LIN {X 0,Y 357.661,Z 442.016,A -85,B 0,C 180,E1 -17550,E2 -17550} C_VEL
LIN {X 0,Y 357.419,Z 441.985,A -85,B 0,C 180,E1 -17551.127,E2 -17551.127} C_VEL
LIN {X 0,Y 356.749,Z 441.848,A -85,B 0,C 180,E1 -17552.258,E2 -17552.258} C_VEL
LIN {X 0,Y 355.709,Z 441.54,A -85,B 0,C 180,E1 -17553.398,E2 -17553.398} C_VEL
LIN {X 0,Y 354.333,Z 441.001,A -85,B 0,C 180,E1 -17554.55,E2 -17554.55} C_VEL
LIN {X 0,Y 352.777,Z 440.106,A -85,B 0,C 180,E1 -17555.717,E2 -17555.717} C_VEL
LIN {X 0,Y 351.014,Z 438.819,A -85,B 0,C 180,E1 -17556.9,E2 -17556.9} C_VEL
LIN {X 0,Y 348.295,Z 436.243,A -85,B 0,C 180,E1 -17558.613,E2 -17558.613} C_VEL
LIN {X 0,Y 346.111,Z 434.166,A -85,B 0,C 180,E1 -17559.779,E2 -17559.779} C_VEL
LIN {X 0,Y 342.714,Z 431.618,A -85,B 0,C 180,E1 -17561.14,E2 -17561.14} C_VEL
LIN {X 0,Y 338.593,Z 427.938,A -85,B 0,C 180,E1 -17562.698,E2 -17562.698} C_VEL
LIN {X 0,Y 333.67,Z 423.547,A -85,B 0,C 180,E1 -17564.333,E2 -17564.333} C_VEL
LIN {X 0,Y 327.334,Z 417.343,A -85,B 0,C 180,E1 -17566.207,E2 -17566.207} C_VEL
LIN {X 0,Y 321.069,Z 411.064,A -85,B 0,C 180,E1 -17567.845,E2 -17567.845} C_VEL
LIN {X 0,Y 314.685,Z 404.327,A -85,B 0,C 180,E1 -17569.339,E2 -17569.339} C_VEL
LIN {X 0,Y 306.772,Z 395.528,A -85,B 0,C 180,E1 -17571.006,E2 -17571.006} C_VEL
LIN {X 0,Y 297.489,Z 384.138,A -85,B 0,C 180,E1 -17572.878,E2 -17572.878} C_VEL
LIN {X 0,Y 291.289,Z 375.491,A -85,B 0,C 180,E1 -17574.11,E2 -17574.11} C_VEL
LIN {X 0,Y 286.082,Z 366.576,A -85,B 0,C 180,E1 -17575.163,E2 -17575.163} C_VEL
LIN {X 0,Y 281.303,Z 356.248,A -85,B 0,C 180,E1 -17576.119,E2 -17576.119} C_VEL
LIN {X 0,Y 277.576,Z 348.553,A -85,B 0,C 180,E1 -17576.746,E2 -17576.746} C_VEL
LIN {X 0,Y 277.359,Z 347.437,A -85,B 0,C 180,E1 -17576.824,E2 -17576.824} C_VEL
LIN {X 0,Y 277.268,Z 347.449,A -85,B 0,C 180,E1 -17580.482,E2 -17580.482} C_VEL
LIN {X 0,Y 277.251,Z 347.451,A -85,B 0,C 180,E1 -17583.895,E2 -17583.895} C_VEL
LIN {X 0,Y 277.286,Z 347.444,A -85,B 0,C 180,E1 -17587.466,E2 -17587.466} C_VEL
LIN {X 0,Y 277.238,Z 347.449,A -85,B 0,C 180,E1 -17591.231,E2 -17591.231} C_VEL
LIN {X 0,Y 277.248,Z 347.448,A -85,B 0,C 180,E1 -17595.216,E2 -17595.216} C_VEL
LIN {X 0,Y 277.292,Z 347.445,A -85,B 0,C 180,E1 -17599.495,E2 -17599.495} C_VEL
LIN {X 0,Y 277.288,Z 347.443,A -85,B 0,C 180,E1 -17602.535,E2 -17602.535} C_VEL
LIN {X 0,Y 277.252,Z 347.448,A -85,B 0,C 180,E1 -17606.106,E2 -17606.106} C_VEL
LIN {X 0,Y 277.259,Z 347.45,A -85,B 0,C 180,E1 -17609.539,E2 -17609.539} C_VEL
LIN {X 0,Y 277.359,Z 347.435,A -85,B 0,C 180,E1 -17612.865,E2 -17612.865} C_VEL
LIN {X 0,Y 277.295,Z 347.441,A -85,B 0,C 180,E1 -17616.077,E2 -17616.077} C_VEL
LIN {X 0,Y 277.343,Z 347.433,A -85,B 0,C 180,E1 -17620.767,E2 -17620.767} C_VEL
LIN {X 0,Y 277.433,Z 347.425,A -85,B 0,C 180,E1 -17625.327,E2 -17625.327} C_VEL
LIN {X 0,Y 277.506,Z 347.413,A -85,B 0,C 180,E1 -17629.79,E2 -17629.79} C_VEL
LIN {X 0,Y 277.648,Z 347.4,A -85,B 0,C 180,E1 -17632.73,E2 -17632.73} C_VEL
LIN {X 0,Y 277.82,Z 347.363,A -85,B 0,C 180,E1 -17638.551,E2 -17638.551} C_VEL
LIN {X 0,Y 277.821,Z 347.375,A -85,B 0,C 180,E1 -17641.45,E2 -17641.45} C_VEL
LIN {X 0,Y 277.649,Z 347.399,A -85,B 0,C 180,E1 -17647.272,E2 -17647.272} C_VEL
LIN {X 0,Y 277.507,Z 347.418,A -85,B 0,C 180,E1 -17650.212,E2 -17650.212} C_VEL
LIN {X 0,Y 277.41,Z 347.432,A -85,B 0,C 180,E1 -17654.676,E2 -17654.676} C_VEL
LIN {X 0,Y 277.324,Z 347.439,A -85,B 0,C 180,E1 -17659.236,E2 -17659.236} C_VEL
LIN {X 0,Y 277.298,Z 347.446,A -85,B 0,C 180,E1 -17663.924,E2 -17663.924} C_VEL
LIN {X 0,Y 277.306,Z 347.44,A -85,B 0,C 180,E1 -17666.283,E2 -17666.283} C_VEL
LIN {X 0,Y 276.643,Z 347.527,A -85,B 0,C 180,E1 -17667.495,E2 -17667.495} C_VEL
LIN {X 0,Y 273.723,Z 347.889,A -85,B 0,C 180,E1 -17669.467,E2 -17669.467} C_VEL
LIN {X 0,Y 271.283,Z 348.334,A -85,B 0,C 180,E1 -17671.069,E2 -17671.069} C_VEL
LIN {X 0,Y 270.308,Z 348.795,A -85,B 0,C 180,E1 -17672.309,E2 -17672.309} C_VEL
LIN {X 0,Y 270.268,Z 348.983,A -85,B 0,C 180,E1 -17672.729,E2 -17672.729} C_VEL
LIN {X 0,Y 270.568,Z 351.115,A -85,B 0,C 180,E1 -17676.687,E2 -17676.687} C_VEL
LIN {X 0,Y 270.931,Z 353.364,A -85,B 0,C 180,E1 -17680.43,E2 -17680.43} C_VEL
LIN {X 0,Y 271.228,Z 355.986,A -85,B 0,C 180,E1 -17684.397,E2 -17684.397} C_VEL
LIN {X 0,Y 271.177,Z 358.336,A -85,B 0,C 180,E1 -17687.637,E2 -17687.637} C_VEL
LIN {X 0,Y 270.855,Z 361.072,A -85,B 0,C 180,E1 -17691.118,E2 -17691.118} C_VEL
LIN {X 0,Y 270.211,Z 364.37,A -85,B 0,C 180,E1 -17695.096,E2 -17695.096} C_VEL
LIN {X 0,Y 269.608,Z 368.108,A -85,B 0,C 180,E1 -17699.343,E2 -17699.343} C_VEL
LIN {X 0,Y 269.108,Z 371.071,A -85,B 0,C 180,E1 -17702.655,E2 -17702.655} C_VEL
LIN {X 0,Y 269.855,Z 374.098,A -85,B 0,C 180,E1 -17702.867,E2 -17702.867} C_VEL
LIN {X 0,Y 273.605,Z 387.988,A -85,B 0,C 180,E1 -17704.108,E2 -17704.108} C_VEL
LIN {X 0,Y 275.578,Z 397.942,A -85,B 0,C 180,E1 -17705.138,E2 -17705.138} C_VEL
LIN {X 0,Y 276.733,Z 406.314,A -85,B 0,C 180,E1 -17706.103,E2 -17706.103} C_VEL
LIN {X 0,Y 277.56,Z 416.03,A -85,B 0,C 180,E1 -17707.392,E2 -17707.392} C_VEL
LIN {X 0,Y 277.591,Z 422.084,A -85,B 0,C 180,E1 -17708.268,E2 -17708.268} C_VEL
LIN {X 0,Y 275.683,Z 432.23,A -85,B 0,C 180,E1 -17709.87,E2 -17709.87} C_VEL
LIN {X 0,Y 274.223,Z 439.743,A -85,B 0,C 180,E1 -17711.316,E2 -17711.316} C_VEL
LIN {X 0,Y 272.724,Z 447.572,A -85,B 0,C 180,E1 -17713.148,E2 -17713.148} C_VEL
LIN {X 0,Y 271.411,Z 454.11,A -85,B 0,C 180,E1 -17714.993,E2 -17714.993} C_VEL
LIN {X 0,Y 270.443,Z 458.61,A -85,B 0,C 180,E1 -17716.474,E2 -17716.474} C_VEL
LIN {X 0,Y 269.43,Z 464.105,A -85,B 0,C 180,E1 -17718.718,E2 -17718.718} C_VEL
LIN {X 0,Y 268.75,Z 468.433,A -85,B 0,C 180,E1 -17720.973,E2 -17720.973} C_VEL
LIN {X 0,Y 268.431,Z 470.802,A -85,B 0,C 180,E1 -17722.478,E2 -17722.478} C_VEL
LIN {X 0,Y 268.181,Z 473.429,A -85,B 0,C 180,E1 -17724.775,E2 -17724.775} C_VEL
LIN {X 0,Y 268.169,Z 475.056,A -85,B 0,C 180,E1 -17726.995,E2 -17726.995} C_VEL
LIN {X 0,Y 268.184,Z 475.647,A -85,B 0,C 180,E1 -17728.498,E2 -17728.498} C_VEL
LIN {X 0,Y 268.184,Z 475.647,A -85,B 0,C 180,E1 -17731.502,E2 -17731.502} C_VEL
LIN {X 0,Y 268.168,Z 475.056,A -85,B 0,C 180,E1 -17733.005,E2 -17733.005} C_VEL
LIN {X 0,Y 268.227,Z 472.603,A -85,B 0,C 180,E1 -17736.016,E2 -17736.016} C_VEL
LIN {X 0,Y 268.565,Z 469.651,A -85,B 0,C 180,E1 -17738.275,E2 -17738.275} C_VEL
LIN {X 0,Y 269.197,Z 465.66,A -85,B 0,C 180,E1 -17740.53,E2 -17740.53} C_VEL
LIN {X 0,Y 270.047,Z 460.526,A -85,B 0,C 180,E1 -17742.78,E2 -17742.78} C_VEL
LIN {X 0,Y 271.136,Z 455.265,A -85,B 0,C 180,E1 -17744.639,E2 -17744.639} C_VEL
LIN {X 0,Y 272.175,Z 450.324,A -85,B 0,C 180,E1 -17746.116,E2 -17746.116} C_VEL
LIN {X 0,Y 273.369,Z 444.625,A -85,B 0,C 180,E1 -17747.582,E2 -17747.582} C_VEL
LIN {X 0,Y 274.872,Z 436.066,A -85,B 0,C 180,E1 -17749.414,E2 -17749.414} C_VEL
LIN {X 0,Y 276.471,Z 427.889,A -85,B 0,C 180,E1 -17750.848,E2 -17750.848} C_VEL
LIN {X 0,Y 277.757,Z 420.73,A -85,B 0,C 180,E1 -17751.914,E2 -17751.914} C_VEL
LIN {X 0,Y 277.247,Z 411.653,A -85,B 0,C 180,E1 -17753.206,E2 -17753.206} C_VEL
LIN {X 0,Y 276.147,Z 401.415,A -85,B 0,C 180,E1 -17754.465,E2 -17754.465} C_VEL
LIN {X 0,Y 274.464,Z 391.943,A -85,B 0,C 180,E1 -17755.495,E2 -17755.495} C_VEL
LIN {X 0,Y 271.783,Z 380.805,A -85,B 0,C 180,E1 -17756.553,E2 -17756.553} C_VEL
LIN {X 0,Y 269.109,Z 371.049,A -85,B 0,C 180,E1 -17757.383,E2 -17757.383} C_VEL
LIN {X 0,Y 269.703,Z 367.344,A -85,B 0,C 180,E1 -17761.41,E2 -17761.41} C_VEL
LIN {X 0,Y 270.228,Z 364.33,A -85,B 0,C 180,E1 -17764.901,E2 -17764.901} C_VEL
LIN {X 0,Y 270.855,Z 361.042,A -85,B 0,C 180,E1 -17768.882,E2 -17768.882} C_VEL
LIN {X 0,Y 271.18,Z 358.333,A -85,B 0,C 180,E1 -17772.363,E2 -17772.363} C_VEL
LIN {X 0,Y 271.228,Z 355.975,A -85,B 0,C 180,E1 -17775.603,E2 -17775.603} C_VEL
LIN {X 0,Y 270.927,Z 353.357,A -85,B 0,C 180,E1 -17779.569,E2 -17779.569} C_VEL
LIN {X 0,Y 270.546,Z 350.92,A -85,B 0,C 180,E1 -17783.638,E2 -17783.638} C_VEL
LIN {X 0,Y 270.314,Z 349.153,A -85,B 0,C 180,E1 -17786.907,E2 -17786.907} C_VEL
LIN {X 0,Y 270.202,Z 348.332,A -85,B 0,C 180,E1 -17789.13,E2 -17789.13} C_VEL
LIN {X 0,Y 270.265,Z 348.321,A -85,B 0,C 180,E1 -17792.145,E2 -17792.145} C_VEL
LIN {X 0,Y 270.239,Z 348.325,A -85,B 0,C 180,E1 -17795.537,E2 -17795.537} C_VEL
LIN {X 0,Y 270.261,Z 348.32,A -85,B 0,C 180,E1 -17800.241,E2 -17800.241} C_VEL
LIN {X 0,Y 270.377,Z 348.305,A -85,B 0,C 180,E1 -17804.933,E2 -17804.933} C_VEL
LIN {X 0,Y 270.442,Z 348.3,A -85,B 0,C 180,E1 -17809.518,E2 -17809.518} C_VEL
LIN {X 0,Y 270.608,Z 348.275,A -85,B 0,C 180,E1 -17812.538,E2 -17812.538} C_VEL
LIN {X 0,Y 270.787,Z 348.251,A -85,B 0,C 180,E1 -17818.512,E2 -17818.512} C_VEL
LIN {X 0,Y 270.786,Z 348.238,A -85,B 0,C 180,E1 -17821.486,E2 -17821.486} C_VEL
LIN {X 0,Y 270.607,Z 348.276,A -85,B 0,C 180,E1 -17827.46,E2 -17827.46} C_VEL
LIN {X 0,Y 270.441,Z 348.294,A -85,B 0,C 180,E1 -17830.48,E2 -17830.48} C_VEL
LIN {X 0,Y 270.402,Z 348.301,A -85,B 0,C 180,E1 -17835.064,E2 -17835.064} C_VEL
LIN {X 0,Y 270.3,Z 348.309,A -85,B 0,C 180,E1 -17839.755,E2 -17839.755} C_VEL
LIN {X 0,Y 270.236,Z 348.321,A -85,B 0,C 180,E1 -17844.588,E2 -17844.588} C_VEL
LIN {X 0,Y 270.27,Z 348.318,A -85,B 0,C 180,E1 -17847.908,E2 -17847.908} C_VEL
LIN {X 0,Y 270.182,Z 348.328,A -85,B 0,C 180,E1 -17851.347,E2 -17851.347} C_VEL
LIN {X 0,Y 270.213,Z 348.325,A -85,B 0,C 180,E1 -17854.903,E2 -17854.903} C_VEL
LIN {X 0,Y 270.219,Z 348.325,A -85,B 0,C 180,E1 -17858.716,E2 -17858.716} C_VEL
LIN {X 0,Y 270.22,Z 348.325,A -85,B 0,C 180,E1 -17862.548,E2 -17862.548} C_VEL
LIN {X 0,Y 270.201,Z 348.326,A -85,B 0,C 180,E1 -17866.742,E2 -17866.742} C_VEL
LIN {X 0,Y 270.234,Z 348.323,A -85,B 0,C 180,E1 -17869.445,E2 -17869.445} C_VEL
LIN {X 0,Y 270.254,Z 348.323,A -85,B 0,C 180,E1 -17873.721,E2 -17873.721} C_VEL
LIN {X 0,Y 270.201,Z 348.327,A -85,B 0,C 180,E1 -17876.892,E2 -17876.892} C_VEL
LIN {X 0,Y 270.225,Z 348.325,A -85,B 0,C 180,E1 -17880.386,E2 -17880.386} C_VEL
LIN {X 0,Y 270.294,Z 348.316,A -85,B 0,C 180,E1 -17882.439,E2 -17882.439} C_VEL
LIN {X 0,Y 271.439,Z 351.352,A -85,B 0,C 180,E1 -17882.676,E2 -17882.676} C_VEL
LIN {X 0,Y 277.296,Z 363.887,A -85,B 0,C 180,E1 -17883.812,E2 -17883.812} C_VEL
LIN {X 0,Y 281.707,Z 373.081,A -85,B 0,C 180,E1 -17884.818,E2 -17884.818} C_VEL
LIN {X 0,Y 287.268,Z 382.022,A -85,B 0,C 180,E1 -17886.046,E2 -17886.046} C_VEL
LIN {X 0,Y 294.883,Z 392.376,A -85,B 0,C 180,E1 -17887.714,E2 -17887.714} C_VEL
LIN {X 0,Y 304.139,Z 403.208,A -85,B 0,C 180,E1 -17889.72,E2 -17889.72} C_VEL
LIN {X 0,Y 312.672,Z 412.496,A -85,B 0,C 180,E1 -17891.659,E2 -17891.659} C_VEL
LIN {X 0,Y 318.129,Z 418.133,A -85,B 0,C 180,E1 -17893.013,E2 -17893.013} C_VEL
LIN {X 0,Y 324.259,Z 424.016,A -85,B 0,C 180,E1 -17894.652,E2 -17894.652} C_VEL
LIN {X 0,Y 330.015,Z 429.444,A -85,B 0,C 180,E1 -17896.452,E2 -17896.452} C_VEL
LIN {X 0,Y 334.064,Z 433.208,A -85,B 0,C 180,E1 -17897.856,E2 -17897.856} C_VEL
LIN {X 0,Y 338.743,Z 437.027,A -85,B 0,C 180,E1 -17899.645,E2 -17899.645} C_VEL
LIN {X 0,Y 341.595,Z 439.344,A -85,B 0,C 180,E1 -17900.946,E2 -17900.946} C_VEL
LIN {X 0,Y 344.973,Z 442.584,A -85,B 0,C 180,E1 -17902.979,E2 -17902.979} C_VEL
LIN {X 0,Y 346.753,Z 443.97,A -85,B 0,C 180,E1 -17904.184,E2 -17904.184} C_VEL
LIN {X 0,Y 348.358,Z 444.934,A -85,B 0,C 180,E1 -17905.371,E2 -17905.371} C_VEL
LIN {X 0,Y 349.734,Z 445.541,A -85,B 0,C 180,E1 -17906.544,E2 -17906.544} C_VEL
LIN {X 0,Y 350.851,Z 445.871,A -85,B 0,C 180,E1 -17907.704,E2 -17907.704} C_VEL
LIN {X 0,Y 351.574,Z 446.038,A -85,B 0,C 180,E1 -17908.855,E2 -17908.855} C_VEL
LIN {X 0,Y 351.859,Z 446.067,A -85,B 0,C 180,E1 -17910,E2 -17910} C_VEL
LIN {X 0,Y 351.482,Z 446.032,A -85,B 0,C 180,E1 -17911.274,E2 -17911.274} C_VEL
LIN {X 0,Y 350.849,Z 445.87,A -85,B 0,C 180,E1 -17912.296,E2 -17912.296} C_VEL
LIN {X 0,Y 349.733,Z 445.538,A -85,B 0,C 180,E1 -17913.456,E2 -17913.456} C_VEL
LIN {X 0,Y 348.327,Z 444.962,A -85,B 0,C 180,E1 -17914.629,E2 -17914.629} C_VEL
LIN {X 0,Y 346.319,Z 443.719,A -85,B 0,C 180,E1 -17916.086,E2 -17916.086} C_VEL
LIN {X 0,Y 342.975,Z 440.779,A -85,B 0,C 180,E1 -17918.247,E2 -17918.247} C_VEL
LIN {X 0,Y 340.73,Z 438.553,A -85,B 0,C 180,E1 -17919.498,E2 -17919.498} C_VEL
LIN {X 0,Y 336.656,Z 435.482,A -85,B 0,C 180,E1 -17921.141,E2 -17921.141} C_VEL
LIN {X 0,Y 333.367,Z 432.558,A -85,B 0,C 180,E1 -17922.393,E2 -17922.393} C_VEL
LIN {X 0,Y 328.668,Z 428.285,A -85,B 0,C 180,E1 -17923.979,E2 -17923.979} C_VEL
LIN {X 0,Y 323.209,Z 423.011,A -85,B 0,C 180,E1 -17925.646,E2 -17925.646} C_VEL
LIN {X 0,Y 316.655,Z 416.567,A -85,B 0,C 180,E1 -17927.379,E2 -17927.379} C_VEL
LIN {X 0,Y 309.433,Z 408.961,A -85,B 0,C 180,E1 -17929.098,E2 -17929.098} C_VEL
LIN {X 0,Y 301.031,Z 399.686,A -85,B 0,C 180,E1 -17930.958,E2 -17930.958} C_VEL
LIN {X 0,Y 292.298,Z 388.981,A -85,B 0,C 180,E1 -17932.859,E2 -17932.859} C_VEL
LIN {X 0,Y 286.35,Z 380.71,A -85,B 0,C 180,E1 -17934.155,E2 -17934.155} C_VEL
LIN {X 0,Y 280.756,Z 371.178,A -85,B 0,C 180,E1 -17935.405,E2 -17935.405} C_VEL
LIN {X 0,Y 276.156,Z 361.254,A -85,B 0,C 180,E1 -17936.436,E2 -17936.436} C_VEL
LIN {X 0,Y 270.473,Z 349.257,A -85,B 0,C 180,E1 -17937.493,E2 -17937.493} C_VEL
LIN {X 0,Y 270.283,Z 348.318,A -85,B 0,C 180,E1 -17937.591,E2 -17937.591} C_VEL
LIN {X 0,Y 270.181,Z 348.33,A -85,B 0,C 180,E1 -17941.348,E2 -17941.348} C_VEL
LIN {X 0,Y 270.212,Z 348.325,A -85,B 0,C 180,E1 -17944.904,E2 -17944.904} C_VEL
LIN {X 0,Y 270.219,Z 348.324,A -85,B 0,C 180,E1 -17948.717,E2 -17948.717} C_VEL
LIN {X 0,Y 270.199,Z 348.326,A -85,B 0,C 180,E1 -17952.553,E2 -17952.553} C_VEL
LIN {X 0,Y 270.211,Z 348.324,A -85,B 0,C 180,E1 -17956.74,E2 -17956.74} C_VEL
LIN {X 0,Y 270.243,Z 348.323,A -85,B 0,C 180,E1 -17959.448,E2 -17959.448} C_VEL
LIN {X 0,Y 270.255,Z 348.322,A -85,B 0,C 180,E1 -17963.722,E2 -17963.722} C_VEL
LIN {X 0,Y 270.202,Z 348.325,A -85,B 0,C 180,E1 -17966.893,E2 -17966.893} C_VEL
LIN {X 0,Y 270.227,Z 348.323,A -85,B 0,C 180,E1 -17970.387,E2 -17970.387} C_VEL
LIN {X 0,Y 270.261,Z 348.318,A -85,B 0,C 180,E1 -17973.765,E2 -17973.765} C_VEL
LIN {X 0,Y 270.208,Z 348.326,A -85,B 0,C 180,E1 -17977.038,E2 -17977.038} C_VEL
LIN {X 0,Y 270.3,Z 348.309,A -85,B 0,C 180,E1 -17980.245,E2 -17980.245} C_VEL
LIN {X 0,Y 270.402,Z 348.301,A -85,B 0,C 180,E1 -17984.936,E2 -17984.936} C_VEL
LIN {X 0,Y 270.441,Z 348.294,A -85,B 0,C 180,E1 -17989.52,E2 -17989.52} C_VEL
LIN {X 0,Y 270.607,Z 348.276,A -85,B 0,C 180,E1 -17992.54,E2 -17992.54} C_VEL
LIN {X 0,Y 270.786,Z 348.238,A -85,B 0,C 180,E1 -17998.514,E2 -17998.514} C_VEL
LIN {X 0,Y 270.787,Z 348.251,A -85,B 0,C 180,E1 -18001.488,E2 -18001.488} C_VEL
LIN {X 0,Y 270.608,Z 348.276,A -85,B 0,C 180,E1 -18007.462,E2 -18007.462} C_VEL
LIN {X 0,Y 270.442,Z 348.3,A -85,B 0,C 180,E1 -18010.482,E2 -18010.482} C_VEL
LIN {X 0,Y 270.377,Z 348.306,A -85,B 0,C 180,E1 -18015.067,E2 -18015.067} C_VEL
LIN {X 0,Y 270.261,Z 348.319,A -85,B 0,C 180,E1 -18019.759,E2 -18019.759} C_VEL
LIN {X 0,Y 270.239,Z 348.325,A -85,B 0,C 180,E1 -18024.59,E2 -18024.59} C_VEL
LIN {X 0,Y 270.271,Z 348.32,A -85,B 0,C 180,E1 -18027.909,E2 -18027.909} C_VEL
LIN {X 0,Y 270.187,Z 348.334,A -85,B 0,C 180,E1 -18031.349,E2 -18031.349} C_VEL
LIN {X 0,Y 270.268,Z 348.983,A -85,B 0,C 180,E1 -18032.729,E2 -18032.729} C_VEL
LIN {X 0,Y 269.722,Z 349.719,A -85,B 0,C 180,E1 -18033.966,E2 -18033.966} C_VEL
LIN {X 0,Y 266.997,Z 351.248,A -85,B 0,C 180,E1 -18035.976,E2 -18035.976} C_VEL
LIN {X 0,Y 264.694,Z 352.535,A -85,B 0,C 180,E1 -18037.609,E2 -18037.609} C_VEL
LIN {X 0,Y 263.801,Z 353.416,A -85,B 0,C 180,E1 -18038.875,E2 -18038.875} C_VEL
LIN {X 0,Y 263.783,Z 353.678,A -85,B 0,C 180,E1 -18039.304,E2 -18039.304} C_VEL
LIN {X 0,Y 264.013,Z 355.221,A -85,B 0,C 180,E1 -18041.81,E2 -18041.81} C_VEL
LIN {X 0,Y 264.157,Z 356.718,A -85,B 0,C 180,E1 -18044.082,E2 -18044.082} C_VEL
LIN {X 0,Y 264.186,Z 358.2,A -85,B 0,C 180,E1 -18046.238,E2 -18046.238} C_VEL
LIN {X 0,Y 264.104,Z 359.695,A -85,B 0,C 180,E1 -18048.297,E2 -18048.297} C_VEL
LIN {X 0,Y 263.868,Z 361.436,A -85,B 0,C 180,E1 -18050.571,E2 -18050.571} C_VEL
LIN {X 0,Y 263.308,Z 364.209,A -85,B 0,C 180,E1 -18054.041,E2 -18054.041} C_VEL
LIN {X 0,Y 262.598,Z 368.332,A -85,B 0,C 180,E1 -18058.919,E2 -18058.919} C_VEL
LIN {X 0,Y 262.112,Z 370.911,A -85,B 0,C 180,E1 -18061.876,E2 -18061.876} C_VEL
LIN {X 0,Y 262.9,Z 373.995,A -85,B 0,C 180,E1 -18062.092,E2 -18062.092} C_VEL
LIN {X 0,Y 266.412,Z 386.666,A -85,B 0,C 180,E1 -18063.265,E2 -18063.265} C_VEL
LIN {X 0,Y 268.686,Z 397.732,A -85,B 0,C 180,E1 -18064.455,E2 -18064.455} C_VEL
LIN {X 0,Y 270.061,Z 407.291,A -85,B 0,C 180,E1 -18065.622,E2 -18065.622} C_VEL
LIN {X 0,Y 270.792,Z 416.062,A -85,B 0,C 180,E1 -18066.83,E2 -18066.83} C_VEL
LIN {X 0,Y 270.965,Z 421.886,A -85,B 0,C 180,E1 -18067.708,E2 -18067.708} C_VEL
LIN {X 0,Y 269.014,Z 432.033,A -85,B 0,C 180,E1 -18069.348,E2 -18069.348} C_VEL
LIN {X 0,Y 267.486,Z 439.547,A -85,B 0,C 180,E1 -18070.827,E2 -18070.827} C_VEL
LIN {X 0,Y 265.919,Z 447.397,A -85,B 0,C 180,E1 -18072.709,E2 -18072.709} C_VEL
LIN {X 0,Y 264.535,Z 453.914,A -85,B 0,C 180,E1 -18074.593,E2 -18074.593} C_VEL
LIN {X 0,Y 263.529,Z 458.414,A -85,B 0,C 180,E1 -18076.112,E2 -18076.112} C_VEL
LIN {X 0,Y 262.434,Z 463.908,A -85,B 0,C 180,E1 -18078.413,E2 -18078.413} C_VEL
LIN {X 0,Y 261.724,Z 468.237,A -85,B 0,C 180,E1 -18080.728,E2 -18080.728} C_VEL
LIN {X 0,Y 261.364,Z 470.605,A -85,B 0,C 180,E1 -18082.273,E2 -18082.273} C_VEL
LIN {X 0,Y 261.088,Z 473.41,A -85,B 0,C 180,E1 -18084.863,E2 -18084.863} C_VEL
LIN {X 0,Y 261.065,Z 474.86,A -85,B 0,C 180,E1 -18086.914,E2 -18086.914} C_VEL
LIN {X 0,Y 261.09,Z 475.452,A -85,B 0,C 180,E1 -18088.458,E2 -18088.458} C_VEL
LIN {X 0,Y 261.127,Z 475.607,A -85,B 0,C 180,E1 -18090,E2 -18090} C_VEL
LIN {X 0,Y 261.09,Z 475.452,A -85,B 0,C 180,E1 -18091.542,E2 -18091.542} C_VEL
LIN {X 0,Y 261.064,Z 474.86,A -85,B 0,C 180,E1 -18093.086,E2 -18093.086} C_VEL
LIN {X 0,Y 261.154,Z 472.407,A -85,B 0,C 180,E1 -18096.18,E2 -18096.18} C_VEL
LIN {X 0,Y 261.53,Z 469.454,A -85,B 0,C 180,E1 -18098.499,E2 -18098.499} C_VEL
LIN {X 0,Y 262.168,Z 465.463,A -85,B 0,C 180,E1 -18100.816,E2 -18100.816} C_VEL
LIN {X 0,Y 263.105,Z 460.33,A -85,B 0,C 180,E1 -18103.123,E2 -18103.123} C_VEL
LIN {X 0,Y 264.257,Z 455.069,A -85,B 0,C 180,E1 -18105.029,E2 -18105.029} C_VEL
LIN {X 0,Y 265.592,Z 448.751,A -85,B 0,C 180,E1 -18106.922,E2 -18106.922} C_VEL
LIN {X 0,Y 266.819,Z 442.798,A -85,B 0,C 180,E1 -18108.426,E2 -18108.426} C_VEL
LIN {X 0,Y 268.156,Z 435.87,A -85,B 0,C 180,E1 -18109.92,E2 -18109.92} C_VEL
LIN {X 0,Y 269.836,Z 427.693,A -85,B 0,C 180,E1 -18111.385,E2 -18111.385} C_VEL
LIN {X 0,Y 270.958,Z 421.886,A -85,B 0,C 180,E1 -18112.293,E2 -18112.293} C_VEL
LIN {X 0,Y 270.422,Z 411.234,A -85,B 0,C 180,E1 -18113.854,E2 -18113.854} C_VEL
LIN {X 0,Y 269.368,Z 401.702,A -85,B 0,C 180,E1 -18115.072,E2 -18115.072} C_VEL
LIN {X 0,Y 267.682,Z 392.269,A -85,B 0,C 180,E1 -18116.146,E2 -18116.146} C_VEL
LIN {X 0,Y 265.249,Z 382.054,A -85,B 0,C 180,E1 -18117.172,E2 -18117.172} C_VEL
LIN {X 0,Y 262.182,Z 371.508,A -85,B 0,C 180,E1 -18118.091,E2 -18118.091} C_VEL
LIN {X 0,Y 262.129,Z 370.896,A -85,B 0,C 180,E1 -18118.151,E2 -18118.151} C_VEL
LIN {X 0,Y 262.604,Z 368.257,A -85,B 0,C 180,E1 -18121.083,E2 -18121.083} C_VEL
LIN {X 0,Y 263.035,Z 365.702,A -85,B 0,C 180,E1 -18124.132,E2 -18124.132} C_VEL
LIN {X 0,Y 263.603,Z 362.677,A -85,B 0,C 180,E1 -18127.822,E2 -18127.822} C_VEL
LIN {X 0,Y 263.902,Z 361.189,A -85,B 0,C 180,E1 -18129.728,E2 -18129.728} C_VEL
LIN {X 0,Y 264.091,Z 359.602,A -85,B 0,C 180,E1 -18131.828,E2 -18131.828} C_VEL
LIN {X 0,Y 264.197,Z 357.961,A -85,B 0,C 180,E1 -18134.09,E2 -18134.09} C_VEL
LIN {X 0,Y 264.127,Z 356.489,A -85,B 0,C 180,E1 -18136.225,E2 -18136.225} C_VEL
LIN {X 0,Y 263.829,Z 353.938,A -85,B 0,C 180,E1 -18140.258,E2 -18140.258} C_VEL
LIN {X 0,Y 263.49,Z 351.738,A -85,B 0,C 180,E1 -18144.069,E2 -18144.069} C_VEL
LIN {X 0,Y 263.218,Z 349.845,A -85,B 0,C 180,E1 -18147.723,E2 -18147.723} C_VEL
LIN {X 0,Y 263.143,Z 349.211,A -85,B 0,C 180,E1 -18149.505,E2 -18149.505} C_VEL
LIN {X 0,Y 263.192,Z 349.201,A -85,B 0,C 180,E1 -18153.002,E2 -18153.002} C_VEL
LIN {X 0,Y 263.155,Z 349.206,A -85,B 0,C 180,E1 -18156.383,E2 -18156.383} C_VEL
LIN {X 0,Y 263.239,Z 349.198,A -85,B 0,C 180,E1 -18159.691,E2 -18159.691} C_VEL
LIN {X 0,Y 263.324,Z 349.183,A -85,B 0,C 180,E1 -18164.52,E2 -18164.52} C_VEL
LIN {X 0,Y 263.374,Z 349.179,A -85,B 0,C 180,E1 -18169.234,E2 -18169.234} C_VEL
LIN {X 0,Y 263.57,Z 349.152,A -85,B 0,C 180,E1 -18172.337,E2 -18172.337} C_VEL
LIN {X 0,Y 263.751,Z 349.128,A -85,B 0,C 180,E1 -18178.472,E2 -18178.472} C_VEL
LIN {X 0,Y 263.751,Z 349.112,A -85,B 0,C 180,E1 -18181.526,E2 -18181.526} C_VEL
LIN {X 0,Y 263.569,Z 349.152,A -85,B 0,C 180,E1 -18187.661,E2 -18187.661} C_VEL
LIN {X 0,Y 263.373,Z 349.176,A -85,B 0,C 180,E1 -18190.765,E2 -18190.765} C_VEL
LIN {X 0,Y 263.35,Z 349.178,A -85,B 0,C 180,E1 -18195.477,E2 -18195.477} C_VEL
LIN {X 0,Y 263.261,Z 349.187,A -85,B 0,C 180,E1 -18200.306,E2 -18200.306} C_VEL
LIN {X 0,Y 263.192,Z 349.197,A -85,B 0,C 180,E1 -18205.292,E2 -18205.292} C_VEL
LIN {X 0,Y 263.178,Z 349.203,A -85,B 0,C 180,E1 -18208.729,E2 -18208.729} C_VEL
LIN {X 0,Y 263.131,Z 349.21,A -85,B 0,C 180,E1 -18212.287,E2 -18212.287} C_VEL
LIN {X 0,Y 263.187,Z 349.201,A -85,B 0,C 180,E1 -18215.977,E2 -18215.977} C_VEL
LIN {X 0,Y 263.158,Z 349.206,A -85,B 0,C 180,E1 -18219.862,E2 -18219.862} C_VEL
LIN {X 0,Y 263.143,Z 349.208,A -85,B 0,C 180,E1 -18223.979,E2 -18223.979} C_VEL
LIN {X 0,Y 263.147,Z 349.206,A -85,B 0,C 180,E1 -18228.4,E2 -18228.4} C_VEL
LIN {X 0,Y 263.185,Z 349.203,A -85,B 0,C 180,E1 -18232.108,E2 -18232.108} C_VEL
LIN {X 0,Y 263.18,Z 349.204,A -85,B 0,C 180,E1 -18235.89,E2 -18235.89} C_VEL
LIN {X 0,Y 263.147,Z 349.208,A -85,B 0,C 180,E1 -18239.507,E2 -18239.507} C_VEL
LIN {X 0,Y 263.221,Z 349.341,A -85,B 0,C 180,E1 -18241.678,E2 -18241.678} C_VEL
LIN {X 0,Y 264.215,Z 352.037,A -85,B 0,C 180,E1 -18241.877,E2 -18241.877} C_VEL
LIN {X 0,Y 269.892,Z 363.561,A -85,B 0,C 180,E1 -18243.004,E2 -18243.004} C_VEL
LIN {X 0,Y 273.726,Z 372.58,A -85,B 0,C 180,E1 -18243.977,E2 -18243.977} C_VEL
LIN {X 0,Y 278.691,Z 381.703,A -85,B 0,C 180,E1 -18245.207,E2 -18245.207} C_VEL
LIN {X 0,Y 285.234,Z 391.448,A -85,B 0,C 180,E1 -18246.782,E2 -18246.782} C_VEL
LIN {X 0,Y 293.941,Z 402.275,A -85,B 0,C 180,E1 -18248.821,E2 -18248.821} C_VEL
LIN {X 0,Y 304.276,Z 413.649,A -85,B 0,C 180,E1 -18251.259,E2 -18251.259} C_VEL
LIN {X 0,Y 311.129,Z 420.736,A -85,B 0,C 180,E1 -18252.923,E2 -18252.923} C_VEL
LIN {X 0,Y 317.486,Z 426.885,A -85,B 0,C 180,E1 -18254.595,E2 -18254.595} C_VEL
LIN {X 0,Y 322.477,Z 431.795,A -85,B 0,C 180,E1 -18256.129,E2 -18256.129} C_VEL
LIN {X 0,Y 328.767,Z 437.503,A -85,B 0,C 180,E1 -18258.284,E2 -18258.284} C_VEL
LIN {X 0,Y 333.898,Z 441.613,A -85,B 0,C 180,E1 -18260.306,E2 -18260.306} C_VEL
LIN {X 0,Y 336.438,Z 443.87,A -85,B 0,C 180,E1 -18261.592,E2 -18261.592} C_VEL
LIN {X 0,Y 339.515,Z 446.678,A -85,B 0,C 180,E1 -18263.51,E2 -18263.51} C_VEL
LIN {X 0,Y 342.001,Z 448.332,A -85,B 0,C 180,E1 -18265.285,E2 -18265.285} C_VEL
LIN {X 0,Y 343.42,Z 449.029,A -85,B 0,C 180,E1 -18266.48,E2 -18266.48} C_VEL
LIN {X 0,Y 344.647,Z 449.438,A -85,B 0,C 180,E1 -18267.692,E2 -18267.692} C_VEL
LIN {X 0,Y 345.423,Z 449.629,A -85,B 0,C 180,E1 -18268.834,E2 -18268.834} C_VEL
LIN {X 0,Y 345.744,Z 449.672,A -85,B 0,C 180,E1 -18270,E2 -18270} C_VEL
LIN {X 0,Y 345.403,Z 449.639,A -85,B 0,C 180,E1 -18271.166,E2 -18271.166} C_VEL
LIN {X 0,Y 344.618,Z 449.428,A -85,B 0,C 180,E1 -18272.338,E2 -18272.338} C_VEL
LIN {X 0,Y 343.413,Z 449.033,A -85,B 0,C 180,E1 -18273.52,E2 -18273.52} C_VEL
LIN {X 0,Y 341.945,Z 448.373,A -85,B 0,C 180,E1 -18274.716,E2 -18274.716} C_VEL
LIN {X 0,Y 339.497,Z 446.749,A -85,B 0,C 180,E1 -18276.463,E2 -18276.463} C_VEL
LIN {X 0,Y 336.443,Z 443.9,A -85,B 0,C 180,E1 -18278.408,E2 -18278.408} C_VEL
LIN {X 0,Y 333.886,Z 441.61,A -85,B 0,C 180,E1 -18279.694,E2 -18279.694} C_VEL
LIN {X 0,Y 328.715,Z 437.487,A -85,B 0,C 180,E1 -18281.718,E2 -18281.718} C_VEL
LIN {X 0,Y 323.656,Z 432.812,A -85,B 0,C 180,E1 -18283.506,E2 -18283.506} C_VEL
LIN {X 0,Y 318.561,Z 428.016,A -85,B 0,C 180,E1 -18285.068,E2 -18285.068} C_VEL
LIN {X 0,Y 312.055,Z 421.712,A -85,B 0,C 180,E1 -18286.834,E2 -18286.834} C_VEL
LIN {X 0,Y 305.564,Z 415.005,A -85,B 0,C 180,E1 -18288.425,E2 -18288.425} C_VEL
LIN {X 0,Y 297.801,Z 406.6,A -85,B 0,C 180,E1 -18290.271,E2 -18290.271} C_VEL
LIN {X 0,Y 290.44,Z 398.084,A -85,B 0,C 180,E1 -18291.999,E2 -18291.999} C_VEL
LIN {X 0,Y 282.971,Z 388.301,A -85,B 0,C 180,E1 -18293.754,E2 -18293.754} C_VEL
LIN {X 0,Y 276.81,Z 378.531,A -85,B 0,C 180,E1 -18295.248,E2 -18295.248} C_VEL
LIN {X 0,Y 272.048,Z 368.742,A -85,B 0,C 180,E1 -18296.456,E2 -18296.456} C_VEL
LIN {X 0,Y 266.742,Z 356.881,A -85,B 0,C 180,E1 -18297.657,E2 -18297.657} C_VEL
LIN {X 0,Y 263.361,Z 350.047,A -85,B 0,C 180,E1 -18298.283,E2 -18298.283} C_VEL
LIN {X 0,Y 263.197,Z 349.202,A -85,B 0,C 180,E1 -18298.363,E2 -18298.363} C_VEL
LIN {X 0,Y 263.13,Z 349.21,A -85,B 0,C 180,E1 -18302.288,E2 -18302.288} C_VEL
LIN {X 0,Y 263.187,Z 349.203,A -85,B 0,C 180,E1 -18305.978,E2 -18305.978} C_VEL
LIN {X 0,Y 263.152,Z 349.208,A -85,B 0,C 180,E1 -18309.864,E2 -18309.864} C_VEL
LIN {X 0,Y 263.141,Z 349.209,A -85,B 0,C 180,E1 -18313.98,E2 -18313.98} C_VEL
LIN {X 0,Y 263.171,Z 349.203,A -85,B 0,C 180,E1 -18318.395,E2 -18318.395} C_VEL
LIN {X 0,Y 263.186,Z 349.202,A -85,B 0,C 180,E1 -18322.109,E2 -18322.109} C_VEL
LIN {X 0,Y 263.181,Z 349.202,A -85,B 0,C 180,E1 -18325.891,E2 -18325.891} C_VEL
LIN {X 0,Y 263.149,Z 349.207,A -85,B 0,C 180,E1 -18329.508,E2 -18329.508} C_VEL
LIN {X 0,Y 263.191,Z 349.2,A -85,B 0,C 180,E1 -18333.004,E2 -18333.004} C_VEL
LIN {X 0,Y 263.153,Z 349.203,A -85,B 0,C 180,E1 -18336.385,E2 -18336.385} C_VEL
LIN {X 0,Y 263.261,Z 349.187,A -85,B 0,C 180,E1 -18339.694,E2 -18339.694} C_VEL
LIN {X 0,Y 263.35,Z 349.178,A -85,B 0,C 180,E1 -18344.523,E2 -18344.523} C_VEL
LIN {X 0,Y 263.373,Z 349.176,A -85,B 0,C 180,E1 -18349.235,E2 -18349.235} C_VEL
LIN {X 0,Y 263.569,Z 349.152,A -85,B 0,C 180,E1 -18352.339,E2 -18352.339} C_VEL
LIN {X 0,Y 263.751,Z 349.112,A -85,B 0,C 180,E1 -18358.474,E2 -18358.474} C_VEL
LIN {X 0,Y 263.751,Z 349.128,A -85,B 0,C 180,E1 -18361.528,E2 -18361.528} C_VEL
LIN {X 0,Y 263.57,Z 349.152,A -85,B 0,C 180,E1 -18367.663,E2 -18367.663} C_VEL
LIN {X 0,Y 263.374,Z 349.18,A -85,B 0,C 180,E1 -18370.766,E2 -18370.766} C_VEL
LIN {X 0,Y 263.324,Z 349.184,A -85,B 0,C 180,E1 -18375.48,E2 -18375.48} C_VEL
LIN {X 0,Y 263.239,Z 349.197,A -85,B 0,C 180,E1 -18380.309,E2 -18380.309} C_VEL
LIN {X 0,Y 263.194,Z 349.202,A -85,B 0,C 180,E1 -18385.294,E2 -18385.294} C_VEL
LIN {X 0,Y 263.167,Z 349.205,A -85,B 0,C 180,E1 -18388.732,E2 -18388.732} C_VEL
LIN {X 0,Y 263.164,Z 349.361,A -85,B 0,C 180,E1 -18391.287,E2 -18391.287} C_VEL
LIN {X 0,Y 263.374,Z 350.816,A -85,B 0,C 180,E1 -18394.186,E2 -18394.186} C_VEL
LIN {X 0,Y 263.635,Z 352.808,A -85,B 0,C 180,E1 -18397.818,E2 -18397.818} C_VEL
LIN {X 0,Y 263.783,Z 353.678,A -85,B 0,C 180,E1 -18399.304,E2 -18399.304} C_VEL
LIN {X 0,Y 263.294,Z 354.531,A -85,B 0,C 180,E1 -18400.566,E2 -18400.566} C_VEL
LIN {X 0,Y 261.838,Z 355.523,A -85,B 0,C 180,E1 -18401.804,E2 -18401.804} C_VEL
LIN {X 0,Y 258.233,Z 357.637,A -85,B 0,C 180,E1 -18404.286,E2 -18404.286} C_VEL
LIN {X 0,Y 257.185,Z 358.643,A -85,B 0,C 180,E1 -18405.578,E2 -18405.578} C_VEL
LIN {X 0,Y 257.091,Z 358.954,A -85,B 0,C 180,E1 -18406.018,E2 -18406.018} C_VEL
LIN {X 0,Y 256.951,Z 361.046,A -85,B 0,C 180,E1 -18408.972,E2 -18408.972} C_VEL
LIN {X 0,Y 256.436,Z 364.046,A -85,B 0,C 180,E1 -18412.919,E2 -18412.919} C_VEL
LIN {X 0,Y 255.788,Z 367.083,A -85,B 0,C 180,E1 -18416.666,E2 -18416.666} C_VEL
LIN {X 0,Y 255.241,Z 370.068,A -85,B 0,C 180,E1 -18420.289,E2 -18420.289} C_VEL
LIN {X 0,Y 255.131,Z 370.723,A -85,B 0,C 180,E1 -18421.034,E2 -18421.034} C_VEL
LIN {X 0,Y 256.05,Z 374.055,A -85,B 0,C 180,E1 -18421.29,E2 -18421.29} C_VEL
LIN {X 0,Y 259.534,Z 386.537,A -85,B 0,C 180,E1 -18422.505,E2 -18422.505} C_VEL
LIN {X 0,Y 261.853,Z 397.522,A -85,B 0,C 180,E1 -18423.738,E2 -18423.738} C_VEL
LIN {X 0,Y 263.23,Z 406.819,A -85,B 0,C 180,E1 -18424.912,E2 -18424.912} C_VEL
LIN {X 0,Y 264.003,Z 416.09,A -85,B 0,C 180,E1 -18426.233,E2 -18426.233} C_VEL
LIN {X 0,Y 264.176,Z 422.951,A -85,B 0,C 180,E1 -18427.31,E2 -18427.31} C_VEL
LIN {X 0,Y 262.335,Z 431.836,A -85,B 0,C 180,E1 -18428.797,E2 -18428.797} C_VEL
LIN {X 0,Y 260.38,Z 440.974,A -85,B 0,C 180,E1 -18430.692,E2 -18430.692} C_VEL
LIN {X 0,Y 259.101,Z 447.353,A -85,B 0,C 180,E1 -18432.284,E2 -18432.284} C_VEL
LIN {X 0,Y 257.664,Z 453.717,A -85,B 0,C 180,E1 -18434.172,E2 -18434.172} C_VEL
LIN {X 0,Y 256.632,Z 458.218,A -85,B 0,C 180,E1 -18435.731,E2 -18435.731} C_VEL
LIN {X 0,Y 255.451,Z 463.711,A -85,B 0,C 180,E1 -18438.092,E2 -18438.092} C_VEL
LIN {X 0,Y 254.681,Z 468.04,A -85,B 0,C 180,E1 -18440.47,E2 -18440.47} C_VEL
LIN {X 0,Y 254.322,Z 470.409,A -85,B 0,C 180,E1 -18442.058,E2 -18442.058} C_VEL
LIN {X 0,Y 253.993,Z 473.395,A -85,B 0,C 180,E1 -18444.961,E2 -18444.961} C_VEL
LIN {X 0,Y 253.964,Z 474.664,A -85,B 0,C 180,E1 -18446.827,E2 -18446.827} C_VEL
LIN {X 0,Y 253.997,Z 475.256,A -85,B 0,C 180,E1 -18448.414,E2 -18448.414} C_VEL
LIN {X 0,Y 254.054,Z 475.412,A -85,B 0,C 180,E1 -18450,E2 -18450} C_VEL
LIN {X 0,Y 253.997,Z 475.256,A -85,B 0,C 180,E1 -18451.586,E2 -18451.586} C_VEL
LIN {X 0,Y 253.963,Z 474.664,A -85,B 0,C 180,E1 -18453.173,E2 -18453.173} C_VEL
LIN {X 0,Y 254.067,Z 472.21,A -85,B 0,C 180,E1 -18456.353,E2 -18456.353} C_VEL
LIN {X 0,Y 254.487,Z 469.258,A -85,B 0,C 180,E1 -18458.736,E2 -18458.736} C_VEL
LIN {X 0,Y 255.154,Z 465.266,A -85,B 0,C 180,E1 -18461.117,E2 -18461.117} C_VEL
LIN {X 0,Y 256.18,Z 460.134,A -85,B 0,C 180,E1 -18463.485,E2 -18463.485} C_VEL
LIN {X 0,Y 257.39,Z 454.872,A -85,B 0,C 180,E1 -18465.44,E2 -18465.44} C_VEL
LIN {X 0,Y 258.795,Z 448.555,A -85,B 0,C 180,E1 -18467.381,E2 -18467.381} C_VEL
LIN {X 0,Y 260.039,Z 442.601,A -85,B 0,C 180,E1 -18468.924,E2 -18468.924} C_VEL
LIN {X 0,Y 261.471,Z 435.673,A -85,B 0,C 180,E1 -18470.452,E2 -18470.452} C_VEL
LIN {X 0,Y 263.229,Z 427.496,A -85,B 0,C 180,E1 -18471.949,E2 -18471.949} C_VEL
LIN {X 0,Y 264.214,Z 421.685,A -85,B 0,C 180,E1 -18472.893,E2 -18472.893} C_VEL
LIN {X 0,Y 263.63,Z 411.029,A -85,B 0,C 180,E1 -18474.509,E2 -18474.509} C_VEL
LIN {X 0,Y 262.62,Z 401.969,A -85,B 0,C 180,E1 -18475.713,E2 -18475.713} C_VEL
LIN {X 0,Y 260.672,Z 391.531,A -85,B 0,C 180,E1 -18476.949,E2 -18476.949} C_VEL
LIN {X 0,Y 258.116,Z 381.111,A -85,B 0,C 180,E1 -18478.033,E2 -18478.033} C_VEL
LIN {X 0,Y 255.231,Z 371.537,A -85,B 0,C 180,E1 -18478.917,E2 -18478.917} C_VEL
LIN {X 0,Y 255.14,Z 370.744,A -85,B 0,C 180,E1 -18478.965,E2 -18478.965} C_VEL
LIN {X 0,Y 255.582,Z 368.511,A -85,B 0,C 180,E1 -18481.521,E2 -18481.521} C_VEL
LIN {X 0,Y 256.116,Z 365.542,A -85,B 0,C 180,E1 -18485.187,E2 -18485.187} C_VEL
LIN {X 0,Y 256.733,Z 362.539,A -85,B 0,C 180,E1 -18489.022,E2 -18489.022} C_VEL
LIN {X 0,Y 257.061,Z 360.033,A -85,B 0,C 180,E1 -18492.423,E2 -18492.423} C_VEL
LIN {X 0,Y 257.123,Z 358.05,A -85,B 0,C 180,E1 -18495.289,E2 -18495.289} C_VEL
LIN {X 0,Y 256.875,Z 355.724,A -85,B 0,C 180,E1 -18498.956,E2 -18498.956} C_VEL
LIN {X 0,Y 256.537,Z 353.409,A -85,B 0,C 180,E1 -18502.935,E2 -18502.935} C_VEL
LIN {X 0,Y 256.265,Z 351.421,A -85,B 0,C 180,E1 -18506.735,E2 -18506.735} C_VEL
LIN {X 0,Y 256.162,Z 350.529,A -85,B 0,C 180,E1 -18508.581,E2 -18508.581} C_VEL
LIN {X 0,Y 256.128,Z 350.083,A -85,B 0,C 180,E1 -18511.409,E2 -18511.409} C_VEL
LIN {X 0,Y 256.143,Z 350.081,A -85,B 0,C 180,E1 -18515.696,E2 -18515.696} C_VEL
LIN {X 0,Y 256.149,Z 350.079,A -85,B 0,C 180,E1 -18519.103,E2 -18519.103} C_VEL
LIN {X 0,Y 256.259,Z 350.064,A -85,B 0,C 180,E1 -18524.082,E2 -18524.082} C_VEL
LIN {X 0,Y 256.29,Z 350.062,A -85,B 0,C 180,E1 -18527.327,E2 -18527.327} C_VEL
LIN {X 0,Y 256.48,Z 350.035,A -85,B 0,C 180,E1 -18530.56,E2 -18530.56} C_VEL
LIN {X 0,Y 256.485,Z 350.036,A -85,B 0,C 180,E1 -18533.707,E2 -18533.707} C_VEL
LIN {X 0,Y 256.714,Z 350.004,A -85,B 0,C 180,E1 -18538.43,E2 -18538.43} C_VEL
LIN {X 0,Y 256.713,Z 349.988,A -85,B 0,C 180,E1 -18541.568,E2 -18541.568} C_VEL
LIN {X 0,Y 256.537,Z 350.027,A -85,B 0,C 180,E1 -18547.872,E2 -18547.872} C_VEL
LIN {X 0,Y 256.309,Z 350.059,A -85,B 0,C 180,E1 -18551.065,E2 -18551.065} C_VEL
LIN {X 0,Y 256.299,Z 350.056,A -85,B 0,C 180,E1 -18555.914,E2 -18555.914} C_VEL
LIN {X 0,Y 256.161,Z 350.076,A -85,B 0,C 180,E1 -18560.895,E2 -18560.895} C_VEL
LIN {X 0,Y 256.169,Z 350.072,A -85,B 0,C 180,E1 -18565.129,E2 -18565.129} C_VEL
LIN {X 0,Y 256.112,Z 350.081,A -85,B 0,C 180,E1 -18569.599,E2 -18569.599} C_VEL
LIN {X 0,Y 256.083,Z 350.083,A -85,B 0,C 180,E1 -18573.289,E2 -18573.289} C_VEL
LIN {X 0,Y 256.138,Z 350.078,A -85,B 0,C 180,E1 -18577.278,E2 -18577.278} C_VEL
LIN {X 0,Y 256.101,Z 350.082,A -85,B 0,C 180,E1 -18581.193,E2 -18581.193} C_VEL
LIN {X 0,Y 256.073,Z 350.086,A -85,B 0,C 180,E1 -18585.525,E2 -18585.525} C_VEL
LIN {X 0,Y 256.082,Z 350.085,A -85,B 0,C 180,E1 -18588.802,E2 -18588.802} C_VEL
LIN {X 0,Y 256.152,Z 350.077,A -85,B 0,C 180,E1 -18592.871,E2 -18592.871} C_VEL
LIN {X 0,Y 256.082,Z 350.086,A -85,B 0,C 180,E1 -18596.71,E2 -18596.71} C_VEL
LIN {X 0,Y 256.128,Z 350.081,A -85,B 0,C 180,E1 -18600.815,E2 -18600.815} C_VEL
LIN {X 0,Y 257.219,Z 353.081,A -85,B 0,C 180,E1 -18601.072,E2 -18601.072} C_VEL
LIN {X 0,Y 262.346,Z 363.243,A -85,B 0,C 180,E1 -18602.131,E2 -18602.131} C_VEL
LIN {X 0,Y 267.687,Z 375.87,A -85,B 0,C 180,E1 -18603.584,E2 -18603.584} C_VEL
LIN {X 0,Y 271.952,Z 384.085,A -85,B 0,C 180,E1 -18604.753,E2 -18604.753} C_VEL
LIN {X 0,Y 278.075,Z 393.612,A -85,B 0,C 180,E1 -18606.371,E2 -18606.371} C_VEL
LIN {X 0,Y 285.937,Z 403.726,A -85,B 0,C 180,E1 -18608.366,E2 -18608.366} C_VEL
LIN {X 0,Y 295.696,Z 414.561,A -85,B 0,C 180,E1 -18610.808,E2 -18610.808} C_VEL
LIN {X 0,Y 304.803,Z 423.872,A -85,B 0,C 180,E1 -18613.111,E2 -18613.111} C_VEL
LIN {X 0,Y 311.274,Z 430.126,A -85,B 0,C 180,E1 -18614.839,E2 -18614.839} C_VEL
LIN {X 0,Y 316.656,Z 435.33,A -85,B 0,C 180,E1 -18616.491,E2 -18616.491} C_VEL
LIN {X 0,Y 321.2,Z 439.481,A -85,B 0,C 180,E1 -18618.003,E2 -18618.003} C_VEL
LIN {X 0,Y 324.914,Z 442.65,A -85,B 0,C 180,E1 -18619.406,E2 -18619.406} C_VEL
LIN {X 0,Y 327.737,Z 444.856,A -85,B 0,C 180,E1 -18620.544,E2 -18620.544} C_VEL
LIN {X 0,Y 330.65,Z 447.541,A -85,B 0,C 180,E1 -18622.059,E2 -18622.059} C_VEL
LIN {X 0,Y 333.607,Z 450.078,A -85,B 0,C 180,E1 -18623.954,E2 -18623.954} C_VEL
LIN {X 0,Y 335.331,Z 451.205,A -85,B 0,C 180,E1 -18625.191,E2 -18625.191} C_VEL
LIN {X 0,Y 337.727,Z 452.381,A -85,B 0,C 180,E1 -18627.252,E2 -18627.252} C_VEL
LIN {X 0,Y 339.005,Z 452.735,A -85,B 0,C 180,E1 -18628.812,E2 -18628.812} C_VEL
LIN {X 0,Y 339.373,Z 452.795,A -85,B 0,C 180,E1 -18630,E2 -18630} C_VEL
LIN {X 0,Y 338.991,Z 452.74,A -85,B 0,C 180,E1 -18631.188,E2 -18631.188} C_VEL
LIN {X 0,Y 337.727,Z 452.384,A -85,B 0,C 180,E1 -18632.746,E2 -18632.746} C_VEL
LIN {X 0,Y 335.263,Z 451.246,A -85,B 0,C 180,E1 -18634.81,E2 -18634.81} C_VEL
LIN {X 0,Y 332.584,Z 449.341,A -85,B 0,C 180,E1 -18636.702,E2 -18636.702} C_VEL
LIN {X 0,Y 329.516,Z 446.431,A -85,B 0,C 180,E1 -18638.586,E2 -18638.586} C_VEL
LIN {X 0,Y 326.629,Z 444.02,A -85,B 0,C 180,E1 -18639.912,E2 -18639.912} C_VEL
LIN {X 0,Y 321.224,Z 439.478,A -85,B 0,C 180,E1 -18641.996,E2 -18641.996} C_VEL
LIN {X 0,Y 315.517,Z 434.281,A -85,B 0,C 180,E1 -18643.874,E2 -18643.874} C_VEL
LIN {X 0,Y 309.97,Z 428.932,A -85,B 0,C 180,E1 -18645.51,E2 -18645.51} C_VEL
LIN {X 0,Y 301.983,Z 421.062,A -85,B 0,C 180,E1 -18647.611,E2 -18647.611} C_VEL
LIN {X 0,Y 291.937,Z 410.514,A -85,B 0,C 180,E1 -18650.139,E2 -18650.139} C_VEL
LIN {X 0,Y 283.306,Z 400.553,A -85,B 0,C 180,E1 -18652.291,E2 -18652.291} C_VEL
LIN {X 0,Y 276.778,Z 391.705,A -85,B 0,C 180,E1 -18653.971,E2 -18653.971} C_VEL
LIN {X 0,Y 271.356,Z 383.043,A -85,B 0,C 180,E1 -18655.406,E2 -18655.406} C_VEL
LIN {X 0,Y 266.29,Z 372.525,A -85,B 0,C 180,E1 -18656.827,E2 -18656.827} C_VEL
LIN {X 0,Y 260.727,Z 359.691,A -85,B 0,C 180,E1 -18658.236,E2 -18658.236} C_VEL
LIN {X 0,Y 256.365,Z 351.265,A -85,B 0,C 180,E1 -18659.097,E2 -18659.097} C_VEL
LIN {X 0,Y 256.128,Z 350.081,A -85,B 0,C 180,E1 -18659.185,E2 -18659.185} C_VEL
LIN {X 0,Y 256.082,Z 350.086,A -85,B 0,C 180,E1 -18663.29,E2 -18663.29} C_VEL
LIN {X 0,Y 256.137,Z 350.079,A -85,B 0,C 180,E1 -18667.279,E2 -18667.279} C_VEL
LIN {X 0,Y 256.082,Z 350.085,A -85,B 0,C 180,E1 -18671.198,E2 -18671.198} C_VEL
LIN {X 0,Y 256.075,Z 350.086,A -85,B 0,C 180,E1 -18675.526,E2 -18675.526} C_VEL
LIN {X 0,Y 256.101,Z 350.082,A -85,B 0,C 180,E1 -18678.807,E2 -18678.807} C_VEL
LIN {X 0,Y 256.153,Z 350.076,A -85,B 0,C 180,E1 -18682.872,E2 -18682.872} C_VEL
LIN {X 0,Y 256.083,Z 350.083,A -85,B 0,C 180,E1 -18686.711,E2 -18686.711} C_VEL
LIN {X 0,Y 256.137,Z 350.08,A -85,B 0,C 180,E1 -18691.405,E2 -18691.405} C_VEL
LIN {X 0,Y 256.141,Z 350.077,A -85,B 0,C 180,E1 -18695.698,E2 -18695.698} C_VEL
LIN {X 0,Y 256.161,Z 350.076,A -85,B 0,C 180,E1 -18699.105,E2 -18699.105} C_VEL
LIN {X 0,Y 256.299,Z 350.056,A -85,B 0,C 180,E1 -18704.086,E2 -18704.086} C_VEL
LIN {X 0,Y 256.309,Z 350.059,A -85,B 0,C 180,E1 -18708.935,E2 -18708.935} C_VEL
LIN {X 0,Y 256.537,Z 350.027,A -85,B 0,C 180,E1 -18712.128,E2 -18712.128} C_VEL
LIN {X 0,Y 256.713,Z 349.988,A -85,B 0,C 180,E1 -18718.432,E2 -18718.432} C_VEL
LIN {X 0,Y 256.714,Z 350.004,A -85,B 0,C 180,E1 -18721.57,E2 -18721.57} C_VEL
LIN {X 0,Y 256.538,Z 350.029,A -85,B 0,C 180,E1 -18727.874,E2 -18727.874} C_VEL
LIN {X 0,Y 256.309,Z 350.059,A -85,B 0,C 180,E1 -18731.067,E2 -18731.067} C_VEL
LIN {X 0,Y 256.238,Z 350.07,A -85,B 0,C 180,E1 -18734.292,E2 -18734.292} C_VEL
LIN {X 0,Y 256.178,Z 350.074,A -85,B 0,C 180,E1 -18737.565,E2 -18737.565} C_VEL
LIN {X 0,Y 256.143,Z 350.078,A -85,B 0,C 180,E1 -18741.112,E2 -18741.112} C_VEL
LIN {X 0,Y 256.172,Z 350.077,A -85,B 0,C 180,E1 -18745.131,E2 -18745.131} C_VEL
LIN {X 0,Y 256.105,Z 350.084,A -85,B 0,C 180,E1 -18749.602,E2 -18749.602} C_VEL
LIN {X 0,Y 256.184,Z 350.682,A -85,B 0,C 180,E1 -18751.742,E2 -18751.742} C_VEL
LIN {X 0,Y 256.404,Z 352.386,A -85,B 0,C 180,E1 -18755.143,E2 -18755.143} C_VEL
LIN {X 0,Y 256.738,Z 354.691,A -85,B 0,C 180,E1 -18759.301,E2 -18759.301} C_VEL
LIN {X 0,Y 257.039,Z 357.023,A -85,B 0,C 180,E1 -18763.123,E2 -18763.123} C_VEL
LIN {X 0,Y 257.091,Z 358.954,A -85,B 0,C 180,E1 -18766.018,E2 -18766.018} C_VEL
LIN {X 0,Y 256.372,Z 359.934,A -85,B 0,C 180,E1 -18767.304,E2 -18767.304} C_VEL
LIN {X 0,Y 253.364,Z 361.77,A -85,B 0,C 180,E1 -18769.386,E2 -18769.386} C_VEL
LIN {X 0,Y 249.794,Z 364.035,A -85,B 0,C 180,E1 -18771.95,E2 -18771.95} C_VEL
LIN {X 0,Y 249.326,Z 364.748,A -85,B 0,C 180,E1 -18772.846,E2 -18772.846} C_VEL
LIN {X 0,Y 248.892,Z 366.897,A -85,B 0,C 180,E1 -18775.616,E2 -18775.616} C_VEL
LIN {X 0,Y 248.292,Z 369.884,A -85,B 0,C 180,E1 -18779.37,E2 -18779.37} C_VEL
LIN {X 0,Y 248.203,Z 370.644,A -85,B 0,C 180,E1 -18780.154,E2 -18780.154} C_VEL
LIN {X 0,Y 249.062,Z 373.788,A -85,B 0,C 180,E1 -18780.403,E2 -18780.403} C_VEL
LIN {X 0,Y 252.625,Z 386.058,A -85,B 0,C 180,E1 -18781.663,E2 -18781.663} C_VEL
LIN {X 0,Y 255.106,Z 397.637,A -85,B 0,C 180,E1 -18783.023,E2 -18783.023} C_VEL
LIN {X 0,Y 256.515,Z 407.247,A -85,B 0,C 180,E1 -18784.292,E2 -18784.292} C_VEL
LIN {X 0,Y 257.209,Z 416.114,A -85,B 0,C 180,E1 -18785.601,E2 -18785.601} C_VEL
LIN {X 0,Y 257.367,Z 423.897,A -85,B 0,C 180,E1 -18786.887,E2 -18786.887} C_VEL
LIN {X 0,Y 255.724,Z 431.64,A -85,B 0,C 180,E1 -18788.222,E2 -18788.222} C_VEL
LIN {X 0,Y 253.674,Z 440.777,A -85,B 0,C 180,E1 -18790.161,E2 -18790.161} C_VEL
LIN {X 0,Y 252.299,Z 447.297,A -85,B 0,C 180,E1 -18791.833,E2 -18791.833} C_VEL
LIN {X 0,Y 250.81,Z 453.52,A -85,B 0,C 180,E1 -18793.727,E2 -18793.727} C_VEL
LIN {X 0,Y 249.719,Z 458.021,A -85,B 0,C 180,E1 -18795.328,E2 -18795.328} C_VEL
LIN {X 0,Y 248.457,Z 463.514,A -85,B 0,C 180,E1 -18797.752,E2 -18797.752} C_VEL
LIN {X 0,Y 247.653,Z 467.843,A -85,B 0,C 180,E1 -18800.196,E2 -18800.196} C_VEL
LIN {X 0,Y 247.273,Z 470.213,A -85,B 0,C 180,E1 -18801.83,E2 -18801.83} C_VEL
LIN {X 0,Y 247.013,Z 472.014,A -85,B 0,C 180,E1 -18803.465,E2 -18803.465} C_VEL
LIN {X 0,Y 246.867,Z 474.468,A -85,B 0,C 180,E1 -18806.736,E2 -18806.736} C_VEL
LIN {X 0,Y 246.907,Z 475.06,A -85,B 0,C 180,E1 -18808.369,E2 -18808.369} C_VEL
LIN {X 0,Y 246.983,Z 475.217,A -85,B 0,C 180,E1 -18810,E2 -18810} C_VEL
LIN {X 0,Y 246.907,Z 475.06,A -85,B 0,C 180,E1 -18811.631,E2 -18811.631} C_VEL
LIN {X 0,Y 246.866,Z 474.468,A -85,B 0,C 180,E1 -18813.264,E2 -18813.264} C_VEL
LIN {X 0,Y 247.012,Z 472.014,A -85,B 0,C 180,E1 -18816.535,E2 -18816.535} C_VEL
LIN {X 0,Y 247.433,Z 469.061,A -85,B 0,C 180,E1 -18818.988,E2 -18818.988} C_VEL
LIN {X 0,Y 248.159,Z 465.069,A -85,B 0,C 180,E1 -18821.434,E2 -18821.434} C_VEL
LIN {X 0,Y 249.241,Z 459.937,A -85,B 0,C 180,E1 -18823.868,E2 -18823.868} C_VEL
LIN {X 0,Y 250.535,Z 454.676,A -85,B 0,C 180,E1 -18825.873,E2 -18825.873} C_VEL
LIN {X 0,Y 252.021,Z 448.359,A -85,B 0,C 180,E1 -18827.864,E2 -18827.864} C_VEL
LIN {X 0,Y 253.662,Z 440.777,A -85,B 0,C 180,E1 -18829.84,E2 -18829.84} C_VEL
LIN {X 0,Y 255.259,Z 433.558,A -85,B 0,C 180,E1 -18831.396,E2 -18831.396} C_VEL
LIN {X 0,Y 257.142,Z 425.032,A -85,B 0,C 180,E1 -18832.921,E2 -18832.921} C_VEL
LIN {X 0,Y 257.419,Z 421.481,A -85,B 0,C 180,E1 -18833.534,E2 -18833.534} C_VEL
LIN {X 0,Y 256.882,Z 411.132,A -85,B 0,C 180,E1 -18835.156,E2 -18835.156} C_VEL
LIN {X 0,Y 255.867,Z 402.255,A -85,B 0,C 180,E1 -18836.39,E2 -18836.39} C_VEL
LIN {X 0,Y 253.947,Z 391.903,A -85,B 0,C 180,E1 -18837.673,E2 -18837.673} C_VEL
LIN {X 0,Y 251.261,Z 381.14,A -85,B 0,C 180,E1 -18838.853,E2 -18838.853} C_VEL
LIN {X 0,Y 248.279,Z 371.279,A -85,B 0,C 180,E1 -18839.809,E2 -18839.809} C_VEL
LIN {X 0,Y 248.213,Z 370.551,A -85,B 0,C 180,E1 -18839.873,E2 -18839.873} C_VEL
LIN {X 0,Y 248.613,Z 368.361,A -85,B 0,C 180,E1 -18842.487,E2 -18842.487} C_VEL
LIN {X 0,Y 249.208,Z 365.38,A -85,B 0,C 180,E1 -18846.315,E2 -18846.315} C_VEL
LIN {X 0,Y 249.85,Z 362.373,A -85,B 0,C 180,E1 -18850.313,E2 -18850.313} C_VEL
LIN {X 0,Y 250.059,Z 360.452,A -85,B 0,C 180,E1 -18853.05,E2 -18853.05} C_VEL
LIN {X 0,Y 250.093,Z 358.905,A -85,B 0,C 180,E1 -18855.368,E2 -18855.368} C_VEL
LIN {X 0,Y 249.826,Z 356.418,A -85,B 0,C 180,E1 -18859.424,E2 -18859.424} C_VEL
LIN {X 0,Y 249.438,Z 354.026,A -85,B 0,C 180,E1 -18863.723,E2 -18863.723} C_VEL
LIN {X 0,Y 249.175,Z 352.002,A -85,B 0,C 180,E1 -18867.795,E2 -18867.795} C_VEL
LIN {X 0,Y 249.082,Z 351.229,A -85,B 0,C 180,E1 -18869.476,E2 -18869.476} C_VEL
LIN {X 0,Y 249.07,Z 350.961,A -85,B 0,C 180,E1 -18873.161,E2 -18873.161} C_VEL
LIN {X 0,Y 249.061,Z 350.962,A -85,B 0,C 180,E1 -18876.73,E2 -18876.73} C_VEL
LIN {X 0,Y 249.087,Z 350.959,A -85,B 0,C 180,E1 -18880.209,E2 -18880.209} C_VEL
LIN {X 0,Y 249.196,Z 350.946,A -85,B 0,C 180,E1 -18883.618,E2 -18883.618} C_VEL
LIN {X 0,Y 249.252,Z 350.936,A -85,B 0,C 180,E1 -18888.616,E2 -18888.616} C_VEL
LIN {X 0,Y 249.48,Z 350.908,A -85,B 0,C 180,E1 -18891.902,E2 -18891.902} C_VEL
LIN {X 0,Y 249.435,Z 350.914,A -85,B 0,C 180,E1 -18896.769,E2 -18896.769} C_VEL
LIN {X 0,Y 249.721,Z 350.866,A -85,B 0,C 180,E1 -18899.999,E2 -18899.999} C_VEL
LIN {X 0,Y 249.435,Z 350.899,A -85,B 0,C 180,E1 -18903.23,E2 -18903.23} C_VEL
LIN {X 0,Y 249.479,Z 350.906,A -85,B 0,C 180,E1 -18908.096,E2 -18908.096} C_VEL
LIN {X 0,Y 249.252,Z 350.937,A -85,B 0,C 180,E1 -18911.383,E2 -18911.383} C_VEL
LIN {X 0,Y 249.241,Z 350.937,A -85,B 0,C 180,E1 -18916.377,E2 -18916.377} C_VEL
LIN {X 0,Y 249.082,Z 350.956,A -85,B 0,C 180,E1 -18921.518,E2 -18921.518} C_VEL
LIN {X 0,Y 249.116,Z 350.95,A -85,B 0,C 180,E1 -18925.475,E2 -18925.475} C_VEL
LIN {X 0,Y 249.082,Z 350.958,A -85,B 0,C 180,E1 -18928.993,E2 -18928.993} C_VEL
LIN {X 0,Y 249.034,Z 350.966,A -85,B 0,C 180,E1 -18932.424,E2 -18932.424} C_VEL
LIN {X 0,Y 249.073,Z 350.96,A -85,B 0,C 180,E1 -18936.337,E2 -18936.337} C_VEL
LIN {X 0,Y 249.075,Z 350.959,A -85,B 0,C 180,E1 -18940.463,E2 -18940.463} C_VEL
LIN {X 0,Y 249.019,Z 350.964,A -85,B 0,C 180,E1 -18944.874,E2 -18944.874} C_VEL
LIN {X 0,Y 249.049,Z 350.961,A -85,B 0,C 180,E1 -18947.37,E2 -18947.37} C_VEL
LIN {X 0,Y 249.048,Z 350.963,A -85,B 0,C 180,E1 -18951.624,E2 -18951.624} C_VEL
LIN {X 0,Y 249.058,Z 350.963,A -85,B 0,C 180,E1 -18955.642,E2 -18955.642} C_VEL
LIN {X 0,Y 249.064,Z 351.075,A -85,B 0,C 180,E1 -18959.95,E2 -18959.95} C_VEL
LIN {X 0,Y 250.045,Z 353.8,A -85,B 0,C 180,E1 -18960.181,E2 -18960.181} C_VEL
LIN {X 0,Y 255.656,Z 364.633,A -85,B 0,C 180,E1 -18961.408,E2 -18961.408} C_VEL
LIN {X 0,Y 259.989,Z 374.977,A -85,B 0,C 180,E1 -18962.643,E2 -18962.643} C_VEL
LIN {X 0,Y 263.713,Z 383.424,A -85,B 0,C 180,E1 -18963.817,E2 -18963.817} C_VEL
LIN {X 0,Y 268.46,Z 391.958,A -85,B 0,C 180,E1 -18965.237,E2 -18965.237} C_VEL
LIN {X 0,Y 274.799,Z 401.139,A -85,B 0,C 180,E1 -18967.026,E2 -18967.026} C_VEL
LIN {X 0,Y 283.846,Z 411.979,A -85,B 0,C 180,E1 -18969.456,E2 -18969.456} C_VEL
LIN {X 0,Y 293.762,Z 422.398,A -85,B 0,C 180,E1 -18972.097,E2 -18972.097} C_VEL
LIN {X 0,Y 302.662,Z 430.911,A -85,B 0,C 180,E1 -18974.502,E2 -18974.502} C_VEL
LIN {X 0,Y 308.906,Z 436.824,A -85,B 0,C 180,E1 -18976.342,E2 -18976.342} C_VEL
LIN {X 0,Y 315.227,Z 442.546,A -85,B 0,C 180,E1 -18978.425,E2 -18978.425} C_VEL
LIN {X 0,Y 320.649,Z 447.012,A -85,B 0,C 180,E1 -18980.504,E2 -18980.504} C_VEL
LIN {X 0,Y 323.483,Z 449.505,A -85,B 0,C 180,E1 -18981.882,E2 -18981.882} C_VEL
LIN {X 0,Y 326.588,Z 452.227,A -85,B 0,C 180,E1 -18983.823,E2 -18983.823} C_VEL
LIN {X 0,Y 328.419,Z 453.525,A -85,B 0,C 180,E1 -18985.09,E2 -18985.09} C_VEL
LIN {X 0,Y 330.765,Z 454.818,A -85,B 0,C 180,E1 -18986.999,E2 -18986.999} C_VEL
LIN {X 0,Y 332.352,Z 455.327,A -85,B 0,C 180,E1 -18988.788,E2 -18988.788} C_VEL
LIN {X 0,Y 332.762,Z 455.404,A -85,B 0,C 180,E1 -18990,E2 -18990} C_VEL
LIN {X 0,Y 332.342,Z 455.33,A -85,B 0,C 180,E1 -18991.212,E2 -18991.212} C_VEL
LIN {X 0,Y 330.76,Z 454.83,A -85,B 0,C 180,E1 -18992.984,E2 -18992.984} C_VEL
LIN {X 0,Y 328.342,Z 453.556,A -85,B 0,C 180,E1 -18994.912,E2 -18994.912} C_VEL
LIN {X 0,Y 325.586,Z 451.447,A -85,B 0,C 180,E1 -18996.819,E2 -18996.819} C_VEL
LIN {X 0,Y 323.479,Z 449.52,A -85,B 0,C 180,E1 -18998.118,E2 -18998.118} C_VEL
LIN {X 0,Y 320.636,Z 447.037,A -85,B 0,C 180,E1 -18999.482,E2 -18999.482} C_VEL
LIN {X 0,Y 315.232,Z 442.523,A -85,B 0,C 180,E1 -19001.575,E2 -19001.575} C_VEL
LIN {X 0,Y 308.927,Z 436.824,A -85,B 0,C 180,E1 -19003.657,E2 -19003.657} C_VEL
LIN {X 0,Y 302.659,Z 430.922,A -85,B 0,C 180,E1 -19005.496,E2 -19005.496} C_VEL
LIN {X 0,Y 293.762,Z 422.363,A -85,B 0,C 180,E1 -19007.91,E2 -19007.91} C_VEL
LIN {X 0,Y 282.954,Z 411.027,A -85,B 0,C 180,E1 -19010.771,E2 -19010.771} C_VEL
LIN {X 0,Y 273.918,Z 399.994,A -85,B 0,C 180,E1 -19013.217,E2 -19013.217} C_VEL
LIN {X 0,Y 266.992,Z 389.466,A -85,B 0,C 180,E1 -19015.198,E2 -19015.198} C_VEL
LIN {X 0,Y 262.195,Z 380.155,A -85,B 0,C 180,E1 -19016.662,E2 -19016.662} C_VEL
LIN {X 0,Y 257.158,Z 368.02,A -85,B 0,C 180,E1 -19018.192,E2 -19018.192} C_VEL
LIN {X 0,Y 252.145,Z 357.564,A -85,B 0,C 180,E1 -19019.4,E2 -19019.4} C_VEL
LIN {X 0,Y 249.277,Z 352.039,A -85,B 0,C 180,E1 -19019.99,E2 -19019.99} C_VEL
LIN {X 0,Y 249.05,Z 350.964,A -85,B 0,C 180,E1 -19020.113,E2 -19020.113} C_VEL
LIN {X 0,Y 249.058,Z 350.963,A -85,B 0,C 180,E1 -19024.358,E2 -19024.358} C_VEL
LIN {X 0,Y 249.048,Z 350.963,A -85,B 0,C 180,E1 -19028.376,E2 -19028.376} C_VEL
LIN {X 0,Y 249.043,Z 350.961,A -85,B 0,C 180,E1 -19032.802,E2 -19032.802} C_VEL
LIN {X 0,Y 249.06,Z 350.96,A -85,B 0,C 180,E1 -19037.373,E2 -19037.373} C_VEL
LIN {X 0,Y 249.05,Z 350.963,A -85,B 0,C 180,E1 -19041.625,E2 -19041.625} C_VEL
LIN {X 0,Y 249.059,Z 350.963,A -85,B 0,C 180,E1 -19045.643,E2 -19045.643} C_VEL
LIN {X 0,Y 249.05,Z 350.963,A -85,B 0,C 180,E1 -19049.474,E2 -19049.474} C_VEL
LIN {X 0,Y 249.069,Z 350.961,A -85,B 0,C 180,E1 -19053.163,E2 -19053.163} C_VEL
LIN {X 0,Y 249.06,Z 350.959,A -85,B 0,C 180,E1 -19056.732,E2 -19056.732} C_VEL
LIN {X 0,Y 249.107,Z 350.949,A -85,B 0,C 180,E1 -19060.212,E2 -19060.212} C_VEL
LIN {X 0,Y 249.241,Z 350.937,A -85,B 0,C 180,E1 -19063.623,E2 -19063.623} C_VEL
LIN {X 0,Y 249.252,Z 350.937,A -85,B 0,C 180,E1 -19068.617,E2 -19068.617} C_VEL
LIN {X 0,Y 249.479,Z 350.906,A -85,B 0,C 180,E1 -19071.904,E2 -19071.904} C_VEL
LIN {X 0,Y 249.435,Z 350.899,A -85,B 0,C 180,E1 -19076.77,E2 -19076.77} C_VEL
LIN {X 0,Y 249.721,Z 350.866,A -85,B 0,C 180,E1 -19080.001,E2 -19080.001} C_VEL
LIN {X 0,Y 249.435,Z 350.914,A -85,B 0,C 180,E1 -19083.231,E2 -19083.231} C_VEL
LIN {X 0,Y 249.48,Z 350.909,A -85,B 0,C 180,E1 -19088.098,E2 -19088.098} C_VEL
LIN {X 0,Y 249.252,Z 350.937,A -85,B 0,C 180,E1 -19091.384,E2 -19091.384} C_VEL
LIN {X 0,Y 249.196,Z 350.946,A -85,B 0,C 180,E1 -19096.487,E2 -19096.487} C_VEL
LIN {X 0,Y 249.082,Z 350.958,A -85,B 0,C 180,E1 -19101.519,E2 -19101.519} C_VEL
LIN {X 0,Y 249.118,Z 350.956,A -85,B 0,C 180,E1 -19105.476,E2 -19105.476} C_VEL
LIN {X 0,Y 249.075,Z 350.96,A -85,B 0,C 180,E1 -19108.99,E2 -19108.99} C_VEL
LIN {X 0,Y 249.082,Z 351.23,A -85,B 0,C 180,E1 -19110.524,E2 -19110.524} C_VEL
LIN {X 0,Y 249.383,Z 353.475,A -85,B 0,C 180,E1 -19115.189,E2 -19115.189} C_VEL
LIN {X 0,Y 249.62,Z 355.114,A -85,B 0,C 180,E1 -19118.274,E2 -19118.274} C_VEL
LIN {X 0,Y 249.99,Z 357.534,A -85,B 0,C 180,E1 -19122.433,E2 -19122.433} C_VEL
LIN {X 0,Y 250.065,Z 359.806,A -85,B 0,C 180,E1 -19125.972,E2 -19125.972} C_VEL
LIN {X 0,Y 249.849,Z 362.4,A -85,B 0,C 180,E1 -19129.687,E2 -19129.687} C_VEL
LIN {X 0,Y 249.326,Z 364.748,A -85,B 0,C 180,E1 -19132.846,E2 -19132.846} C_VEL
LIN {X 0,Y 248.484,Z 365.49,A -85,B 0,C 180,E1 -19133.721,E2 -19133.721} C_VEL
LIN {X 0,Y 245.39,Z 366.816,A -85,B 0,C 180,E1 -19135.074,E2 -19135.074} C_VEL
LIN {X 0,Y 242.318,Z 368.154,A -85,B 0,C 180,E1 -19136.458,E2 -19136.458} C_VEL
LIN {X 0,Y 241.545,Z 368.916,A -85,B 0,C 180,E1 -19137.371,E2 -19137.371} C_VEL
LIN {X 0,Y 241.263,Z 370.489,A -85,B 0,C 180,E1 -19139.206,E2 -19139.206} C_VEL
LIN {X 0,Y 242.177,Z 373.695,A -85,B 0,C 180,E1 -19139.48,E2 -19139.48} C_VEL
LIN {X 0,Y 246.08,Z 387.132,A -85,B 0,C 180,E1 -19140.954,E2 -19140.954} C_VEL
LIN {X 0,Y 248.262,Z 397.37,A -85,B 0,C 180,E1 -19142.21,E2 -19142.21} C_VEL
LIN {X 0,Y 249.735,Z 407.215,A -85,B 0,C 180,E1 -19143.565,E2 -19143.565} C_VEL
LIN {X 0,Y 250.448,Z 415.681,A -85,B 0,C 180,E1 -19144.861,E2 -19144.861} C_VEL
LIN {X 0,Y 250.597,Z 424.836,A -85,B 0,C 180,E1 -19146.444,E2 -19146.444} C_VEL
LIN {X 0,Y 248.652,Z 433.362,A -85,B 0,C 180,E1 -19148.006,E2 -19148.006} C_VEL
LIN {X 0,Y 246.98,Z 440.581,A -85,B 0,C 180,E1 -19149.599,E2 -19149.599} C_VEL
LIN {X 0,Y 245.66,Z 446.655,A -85,B 0,C 180,E1 -19151.184,E2 -19151.184} C_VEL
LIN {X 0,Y 243.962,Z 453.323,A -85,B 0,C 180,E1 -19153.257,E2 -19153.257} C_VEL
LIN {X 0,Y 242.831,Z 457.825,A -85,B 0,C 180,E1 -19154.902,E2 -19154.902} C_VEL
LIN {X 0,Y 241.483,Z 463.317,A -85,B 0,C 180,E1 -19157.392,E2 -19157.392} C_VEL
LIN {X 0,Y 240.638,Z 467.647,A -85,B 0,C 180,E1 -19159.908,E2 -19159.908} C_VEL
LIN {X 0,Y 240.22,Z 470.016,A -85,B 0,C 180,E1 -19161.589,E2 -19161.589} C_VEL
LIN {X 0,Y 239.956,Z 471.818,A -85,B 0,C 180,E1 -19163.272,E2 -19163.272} C_VEL
LIN {X 0,Y 239.772,Z 474.272,A -85,B 0,C 180,E1 -19166.639,E2 -19166.639} C_VEL
LIN {X 0,Y 239.819,Z 474.865,A -85,B 0,C 180,E1 -19168.321,E2 -19168.321} C_VEL
LIN {X 0,Y 239.891,Z 475.022,A -85,B 0,C 180,E1 -19170,E2 -19170} C_VEL
LIN {X 0,Y 239.818,Z 474.865,A -85,B 0,C 180,E1 -19171.679,E2 -19171.679} C_VEL
LIN {X 0,Y 239.771,Z 474.272,A -85,B 0,C 180,E1 -19173.361,E2 -19173.361} C_VEL
LIN {X 0,Y 239.955,Z 471.818,A -85,B 0,C 180,E1 -19176.728,E2 -19176.728} C_VEL
LIN {X 0,Y 240.4,Z 468.865,A -85,B 0,C 180,E1 -19179.253,E2 -19179.253} C_VEL
LIN {X 0,Y 241.176,Z 464.873,A -85,B 0,C 180,E1 -19181.77,E2 -19181.77} C_VEL
LIN {X 0,Y 242.32,Z 459.74,A -85,B 0,C 180,E1 -19184.272,E2 -19184.272} C_VEL
LIN {X 0,Y 243.692,Z 454.479,A -85,B 0,C 180,E1 -19186.331,E2 -19186.331} C_VEL
LIN {X 0,Y 245.268,Z 448.163,A -85,B 0,C 180,E1 -19188.373,E2 -19188.373} C_VEL
LIN {X 0,Y 246.585,Z 442.207,A -85,B 0,C 180,E1 -19190,E2 -19190} C_VEL
LIN {X 0,Y 248.18,Z 435.281,A -85,B 0,C 180,E1 -19191.601,E2 -19191.601} C_VEL
LIN {X 0,Y 250.076,Z 427.104,A -85,B 0,C 180,E1 -19193.169,E2 -19193.169} C_VEL
LIN {X 0,Y 250.691,Z 423.696,A -85,B 0,C 180,E1 -19193.766,E2 -19193.766} C_VEL
LIN {X 0,Y 250.21,Z 411.943,A -85,B 0,C 180,E1 -19195.737,E2 -19195.737} C_VEL
LIN {X 0,Y 249.159,Z 402.558,A -85,B 0,C 180,E1 -19197.101,E2 -19197.101} C_VEL
LIN {X 0,Y 247.024,Z 391.365,A -85,B 0,C 180,E1 -19198.547,E2 -19198.547} C_VEL
LIN {X 0,Y 244.325,Z 380.645,A -85,B 0,C 180,E1 -19199.772,E2 -19199.772} C_VEL
LIN {X 0,Y 241.327,Z 371.034,A -85,B 0,C 180,E1 -19200.76,E2 -19200.76} C_VEL
LIN {X 0,Y 241.261,Z 370.36,A -85,B 0,C 180,E1 -19200.839,E2 -19200.839} C_VEL
LIN {X 0,Y 241.667,Z 368.203,A -85,B 0,C 180,E1 -19203.542,E2 -19203.542} C_VEL
LIN {X 0,Y 242.328,Z 365.201,A -85,B 0,C 180,E1 -19207.52,E2 -19207.52} C_VEL
LIN {X 0,Y 242.817,Z 362.572,A -85,B 0,C 180,E1 -19211.189,E2 -19211.189} C_VEL
LIN {X 0,Y 243.037,Z 360.726,A -85,B 0,C 180,E1 -19213.949,E2 -19213.949} C_VEL
LIN {X 0,Y 243.004,Z 359.239,A -85,B 0,C 180,E1 -19216.305,E2 -19216.305} C_VEL
LIN {X 0,Y 242.666,Z 356.839,A -85,B 0,C 180,E1 -19220.419,E2 -19220.419} C_VEL
LIN {X 0,Y 242.371,Z 354.649,A -85,B 0,C 180,E1 -19224.553,E2 -19224.553} C_VEL
LIN {X 0,Y 242.118,Z 352.771,A -85,B 0,C 180,E1 -19228.5,E2 -19228.5} C_VEL
LIN {X 0,Y 242.019,Z 351.851,A -85,B 0,C 180,E1 -19230.595,E2 -19230.595} C_VEL
LIN {X 0,Y 242.069,Z 351.834,A -85,B 0,C 180,E1 -19234.182,E2 -19234.182} C_VEL
LIN {X 0,Y 242.025,Z 351.839,A -85,B 0,C 180,E1 -19238.314,E2 -19238.314} C_VEL
LIN {X 0,Y 242.128,Z 351.826,A -85,B 0,C 180,E1 -19243.306,E2 -19243.306} C_VEL
LIN {X 0,Y 242.184,Z 351.816,A -85,B 0,C 180,E1 -19248.279,E2 -19248.279} C_VEL
LIN {X 0,Y 242.427,Z 351.788,A -85,B 0,C 180,E1 -19251.665,E2 -19251.665} C_VEL
LIN {X 0,Y 242.259,Z 351.809,A -85,B 0,C 180,E1 -19255.006,E2 -19255.006} C_VEL
LIN {X 0,Y 242.636,Z 351.757,A -85,B 0,C 180,E1 -19258.339,E2 -19258.339} C_VEL
LIN {X 0,Y 242.636,Z 351.738,A -85,B 0,C 180,E1 -19261.659,E2 -19261.659} C_VEL
LIN {X 0,Y 242.428,Z 351.786,A -85,B 0,C 180,E1 -19266.698,E2 -19266.698} C_VEL
LIN {X 0,Y 242.313,Z 351.796,A -85,B 0,C 180,E1 -19270.021,E2 -19270.021} C_VEL
LIN {X 0,Y 242.166,Z 351.816,A -85,B 0,C 180,E1 -19275.14,E2 -19275.14} C_VEL
LIN {X 0,Y 242.071,Z 351.83,A -85,B 0,C 180,E1 -19278.623,E2 -19278.623} C_VEL
LIN {X 0,Y 242.005,Z 351.839,A -85,B 0,C 180,E1 -19282.18,E2 -19282.18} C_VEL
LIN {X 0,Y 242.065,Z 351.828,A -85,B 0,C 180,E1 -19285.837,E2 -19285.837} C_VEL
LIN {X 0,Y 242.028,Z 351.836,A -85,B 0,C 180,E1 -19289.579,E2 -19289.579} C_VEL
LIN {X 0,Y 241.989,Z 351.839,A -85,B 0,C 180,E1 -19293.49,E2 -19293.49} C_VEL
LIN {X 0,Y 242.01,Z 351.838,A -85,B 0,C 180,E1 -19297.577,E2 -19297.577} C_VEL
LIN {X 0,Y 241.982,Z 351.844,A -85,B 0,C 180,E1 -19301.911,E2 -19301.911} C_VEL
LIN {X 0,Y 241.983,Z 351.842,A -85,B 0,C 180,E1 -19306.558,E2 -19306.558} C_VEL
LIN {X 0,Y 241.985,Z 351.843,A -85,B 0,C 180,E1 -19310.287,E2 -19310.287} C_VEL
LIN {X 0,Y 242.033,Z 351.837,A -85,B 0,C 180,E1 -19314.497,E2 -19314.497} C_VEL
LIN {X 0,Y 241.991,Z 351.842,A -85,B 0,C 180,E1 -19318.967,E2 -19318.967} C_VEL
LIN {X 0,Y 243,Z 354.694,A -85,B 0,C 180,E1 -19319.255,E2 -19319.255} C_VEL
LIN {X 0,Y 248.692,Z 365.546,A -85,B 0,C 180,E1 -19320.576,E2 -19320.576} C_VEL
LIN {X 0,Y 253.479,Z 376.814,A -85,B 0,C 180,E1 -19322.023,E2 -19322.023} C_VEL
LIN {X 0,Y 257.106,Z 385.625,A -85,B 0,C 180,E1 -19323.301,E2 -19323.301} C_VEL
LIN {X 0,Y 260.78,Z 392.765,A -85,B 0,C 180,E1 -19324.527,E2 -19324.527} C_VEL
LIN {X 0,Y 267.033,Z 402.585,A -85,B 0,C 180,E1 -19326.494,E2 -19326.494} C_VEL
LIN {X 0,Y 276.039,Z 413.751,A -85,B 0,C 180,E1 -19329.118,E2 -19329.118} C_VEL
LIN {X 0,Y 285.086,Z 423.161,A -85,B 0,C 180,E1 -19331.637,E2 -19331.637} C_VEL
LIN {X 0,Y 293.94,Z 431.64,A -85,B 0,C 180,E1 -19334.15,E2 -19334.15} C_VEL
LIN {X 0,Y 300.001,Z 436.926,A -85,B 0,C 180,E1 -19335.887,E2 -19335.887} C_VEL
LIN {X 0,Y 306.837,Z 443.099,A -85,B 0,C 180,E1 -19338.104,E2 -19338.104} C_VEL
LIN {X 0,Y 312.532,Z 447.962,A -85,B 0,C 180,E1 -19340.198,E2 -19340.198} C_VEL
LIN {X 0,Y 315.99,Z 450.835,A -85,B 0,C 180,E1 -19341.688,E2 -19341.688} C_VEL
LIN {X 0,Y 319.344,Z 453.775,A -85,B 0,C 180,E1 -19343.683,E2 -19343.683} C_VEL
LIN {X 0,Y 321.253,Z 455.264,A -85,B 0,C 180,E1 -19344.98,E2 -19344.98} C_VEL
LIN {X 0,Y 323.75,Z 456.748,A -85,B 0,C 180,E1 -19346.921,E2 -19346.921} C_VEL
LIN {X 0,Y 325.462,Z 457.32,A -85,B 0,C 180,E1 -19348.763,E2 -19348.763} C_VEL
LIN {X 0,Y 325.953,Z 457.392,A -85,B 0,C 180,E1 -19350,E2 -19350} C_VEL
LIN {X 0,Y 325.454,Z 457.321,A -85,B 0,C 180,E1 -19351.237,E2 -19351.237} C_VEL
LIN {X 0,Y 323.744,Z 456.764,A -85,B 0,C 180,E1 -19353.057,E2 -19353.057} C_VEL
LIN {X 0,Y 321.191,Z 455.27,A -85,B 0,C 180,E1 -19355.021,E2 -19355.021} C_VEL
LIN {X 0,Y 318.518,Z 453.118,A -85,B 0,C 180,E1 -19356.833,E2 -19356.833} C_VEL
LIN {X 0,Y 315.989,Z 450.84,A -85,B 0,C 180,E1 -19358.312,E2 -19358.312} C_VEL
LIN {X 0,Y 312.515,Z 447.992,A -85,B 0,C 180,E1 -19359.796,E2 -19359.796} C_VEL
LIN {X 0,Y 306.876,Z 443.098,A -85,B 0,C 180,E1 -19361.895,E2 -19361.895} C_VEL
LIN {X 0,Y 299.988,Z 436.945,A -85,B 0,C 180,E1 -19364.109,E2 -19364.109} C_VEL
LIN {X 0,Y 291.545,Z 429.349,A -85,B 0,C 180,E1 -19366.549,E2 -19366.549} C_VEL
LIN {X 0,Y 282.535,Z 420.718,A -85,B 0,C 180,E1 -19369.051,E2 -19369.051} C_VEL
LIN {X 0,Y 273.707,Z 411.067,A -85,B 0,C 180,E1 -19371.546,E2 -19371.546} C_VEL
LIN {X 0,Y 265.488,Z 400.353,A -85,B 0,C 180,E1 -19373.985,E2 -19373.985} C_VEL
LIN {X 0,Y 259.643,Z 390.762,A -85,B 0,C 180,E1 -19375.843,E2 -19375.843} C_VEL
LIN {X 0,Y 255.244,Z 381.307,A -85,B 0,C 180,E1 -19377.363,E2 -19377.363} C_VEL
LIN {X 0,Y 250.305,Z 369.066,A -85,B 0,C 180,E1 -19378.981,E2 -19378.981} C_VEL
LIN {X 0,Y 245.034,Z 358.356,A -85,B 0,C 180,E1 -19380.316,E2 -19380.316} C_VEL
LIN {X 0,Y 242.231,Z 352.925,A -85,B 0,C 180,E1 -19380.933,E2 -19380.933} C_VEL
LIN {X 0,Y 241.991,Z 351.842,A -85,B 0,C 180,E1 -19381.033,E2 -19381.033} C_VEL
LIN {X 0,Y 242.026,Z 351.838,A -85,B 0,C 180,E1 -19385.605,E2 -19385.605} C_VEL
LIN {X 0,Y 241.985,Z 351.843,A -85,B 0,C 180,E1 -19389.713,E2 -19389.713} C_VEL
LIN {X 0,Y 241.973,Z 351.844,A -85,B 0,C 180,E1 -19394.192,E2 -19394.192} C_VEL
LIN {X 0,Y 241.982,Z 351.844,A -85,B 0,C 180,E1 -19398.089,E2 -19398.089} C_VEL
LIN {X 0,Y 242.01,Z 351.838,A -85,B 0,C 180,E1 -19402.423,E2 -19402.423} C_VEL
LIN {X 0,Y 241.989,Z 351.839,A -85,B 0,C 180,E1 -19406.51,E2 -19406.51} C_VEL
LIN {X 0,Y 242.035,Z 351.835,A -85,B 0,C 180,E1 -19410.588,E2 -19410.588} C_VEL
LIN {X 0,Y 242.066,Z 351.828,A -85,B 0,C 180,E1 -19414.184,E2 -19414.184} C_VEL
LIN {X 0,Y 242.024,Z 351.836,A -85,B 0,C 180,E1 -19418.314,E2 -19418.314} C_VEL
LIN {X 0,Y 242.162,Z 351.821,A -85,B 0,C 180,E1 -19423.279,E2 -19423.279} C_VEL
LIN {X 0,Y 242.186,Z 351.816,A -85,B 0,C 180,E1 -19428.281,E2 -19428.281} C_VEL
LIN {X 0,Y 242.426,Z 351.786,A -85,B 0,C 180,E1 -19431.666,E2 -19431.666} C_VEL
LIN {X 0,Y 242.258,Z 351.803,A -85,B 0,C 180,E1 -19435.008,E2 -19435.008} C_VEL
LIN {X 0,Y 242.636,Z 351.738,A -85,B 0,C 180,E1 -19438.341,E2 -19438.341} C_VEL
LIN {X 0,Y 242.636,Z 351.757,A -85,B 0,C 180,E1 -19441.661,E2 -19441.661} C_VEL
LIN {X 0,Y 242.432,Z 351.788,A -85,B 0,C 180,E1 -19446.66,E2 -19446.66} C_VEL
LIN {X 0,Y 242.314,Z 351.802,A -85,B 0,C 180,E1 -19450.023,E2 -19450.023} C_VEL
LIN {X 0,Y 242.14,Z 351.824,A -85,B 0,C 180,E1 -19455.143,E2 -19455.143} C_VEL
LIN {X 0,Y 242.05,Z 351.836,A -85,B 0,C 180,E1 -19458.627,E2 -19458.627} C_VEL
LIN {X 0,Y 242.006,Z 351.842,A -85,B 0,C 180,E1 -19462.182,E2 -19462.182} C_VEL
LIN {X 0,Y 242.068,Z 351.836,A -85,B 0,C 180,E1 -19465.839,E2 -19465.839} C_VEL
LIN {X 0,Y 242.035,Z 351.919,A -85,B 0,C 180,E1 -19469.581,E2 -19469.581} C_VEL
LIN {X 0,Y 242.228,Z 353.675,A -85,B 0,C 180,E1 -19473.455,E2 -19473.455} C_VEL
LIN {X 0,Y 242.512,Z 355.716,A -85,B 0,C 180,E1 -19477.488,E2 -19477.488} C_VEL
LIN {X 0,Y 242.879,Z 358.062,A -85,B 0,C 180,E1 -19481.724,E2 -19481.724} C_VEL
LIN {X 0,Y 243.019,Z 359.401,A -85,B 0,C 180,E1 -19483.954,E2 -19483.954} C_VEL
LIN {X 0,Y 243.029,Z 360.915,A -85,B 0,C 180,E1 -19486.3,E2 -19486.3} C_VEL
LIN {X 0,Y 242.642,Z 363.729,A -85,B 0,C 180,E1 -19490.416,E2 -19490.416} C_VEL
LIN {X 0,Y 241.983,Z 366.713,A -85,B 0,C 180,E1 -19494.489,E2 -19494.489} C_VEL
LIN {X 0,Y 241.545,Z 368.916,A -85,B 0,C 180,E1 -19497.371,E2 -19497.371} C_VEL
LIN {X 0,Y 241.458,Z 370.403,A -85,B 0,C 180,E1 -19498.177,E2 -19498.177} C_VEL
LIN {X 0,Y 241.353,Z 372.989,A -85,B 0,C 180,E1 -19498.829,E2 -19498.829} C_VEL
LIN {X 0,Y 241.153,Z 378.032,A -85,B 0,C 180,E1 -19499.557,E2 -19499.557} C_VEL
LIN {X 0,Y 241.067,Z 394.21,A -85,B 0,C 180,E1 -19500.966,E2 -19500.966} C_VEL
LIN {X 0,Y 241.272,Z 396.106,A -85,B 0,C 180,E1 -19501.209,E2 -19501.209} C_VEL
LIN {X 0,Y 242.872,Z 406.122,A -85,B 0,C 180,E1 -19502.632,E2 -19502.632} C_VEL
LIN {X 0,Y 243.702,Z 415.1,A -85,B 0,C 180,E1 -19504.051,E2 -19504.051} C_VEL
LIN {X 0,Y 243.945,Z 424.635,A -85,B 0,C 180,E1 -19505.761,E2 -19505.761} C_VEL
LIN {X 0,Y 242.074,Z 433.166,A -85,B 0,C 180,E1 -19507.376,E2 -19507.376} C_VEL
LIN {X 0,Y 240.299,Z 440.384,A -85,B 0,C 180,E1 -19509.006,E2 -19509.006} C_VEL
LIN {X 0,Y 238.832,Z 446.772,A -85,B 0,C 180,E1 -19510.727,E2 -19510.727} C_VEL
LIN {X 0,Y 237.127,Z 453.126,A -85,B 0,C 180,E1 -19512.76,E2 -19512.76} C_VEL
LIN {X 0,Y 235.952,Z 457.628,A -85,B 0,C 180,E1 -19514.451,E2 -19514.451} C_VEL
LIN {X 0,Y 234.528,Z 463.12,A -85,B 0,C 180,E1 -19517.012,E2 -19517.012} C_VEL
LIN {X 0,Y 233.609,Z 467.45,A -85,B 0,C 180,E1 -19519.601,E2 -19519.601} C_VEL
LIN {X 0,Y 233.188,Z 469.82,A -85,B 0,C 180,E1 -19521.333,E2 -19521.333} C_VEL
LIN {X 0,Y 232.893,Z 471.622,A -85,B 0,C 180,E1 -19523.067,E2 -19523.067} C_VEL
LIN {X 0,Y 232.681,Z 474.076,A -85,B 0,C 180,E1 -19526.537,E2 -19526.537} C_VEL
LIN {X 0,Y 232.732,Z 474.669,A -85,B 0,C 180,E1 -19528.27,E2 -19528.27} C_VEL
LIN {X 0,Y 232.802,Z 474.826,A -85,B 0,C 180,E1 -19530,E2 -19530} C_VEL
LIN {X 0,Y 232.732,Z 474.669,A -85,B 0,C 180,E1 -19531.73,E2 -19531.73} C_VEL
LIN {X 0,Y 232.692,Z 473.391,A -85,B 0,C 180,E1 -19534.647,E2 -19534.647} C_VEL
LIN {X 0,Y 232.892,Z 471.622,A -85,B 0,C 180,E1 -19536.933,E2 -19536.933} C_VEL
LIN {X 0,Y 233.384,Z 468.668,A -85,B 0,C 180,E1 -19539.533,E2 -19539.533} C_VEL
LIN {X 0,Y 234.187,Z 464.676,A -85,B 0,C 180,E1 -19542.126,E2 -19542.126} C_VEL
LIN {X 0,Y 235.419,Z 459.543,A -85,B 0,C 180,E1 -19544.7,E2 -19544.7} C_VEL
LIN {X 0,Y 236.863,Z 454.283,A -85,B 0,C 180,E1 -19546.816,E2 -19546.816} C_VEL
LIN {X 0,Y 238.509,Z 447.966,A -85,B 0,C 180,E1 -19548.913,E2 -19548.913} C_VEL
LIN {X 0,Y 240.28,Z 440.383,A -85,B 0,C 180,E1 -19550.996,E2 -19550.996} C_VEL
LIN {X 0,Y 242.051,Z 433.165,A -85,B 0,C 180,E1 -19552.626,E2 -19552.626} C_VEL
LIN {X 0,Y 243.932,Z 424.634,A -85,B 0,C 180,E1 -19554.24,E2 -19554.24} C_VEL
LIN {X 0,Y 243.72,Z 415.036,A -85,B 0,C 180,E1 -19555.958,E2 -19555.958} C_VEL
LIN {X 0,Y 242.555,Z 403.556,A -85,B 0,C 180,E1 -19557.76,E2 -19557.76} C_VEL
LIN {X 0,Y 240.6,Z 392.693,A -85,B 0,C 180,E1 -19559.24,E2 -19559.24} C_VEL
LIN {X 0,Y 237.521,Z 380.787,A -85,B 0,C 180,E1 -19560.69,E2 -19560.69} C_VEL
LIN {X 0,Y 234.52,Z 371.256,A -85,B 0,C 180,E1 -19561.734,E2 -19561.734} C_VEL
LIN {X 0,Y 234.38,Z 370.164,A -85,B 0,C 180,E1 -19561.871,E2 -19561.871} C_VEL
LIN {X 0,Y 235.099,Z 366.517,A -85,B 0,C 180,E1 -19566.718,E2 -19566.718} C_VEL
LIN {X 0,Y 235.511,Z 364.827,A -85,B 0,C 180,E1 -19569.114,E2 -19569.114} C_VEL
LIN {X 0,Y 235.923,Z 362.049,A -85,B 0,C 180,E1 -19573.248,E2 -19573.248} C_VEL
LIN {X 0,Y 235.93,Z 359.884,A -85,B 0,C 180,E1 -19576.753,E2 -19576.753} C_VEL
LIN {X 0,Y 235.62,Z 357.582,A -85,B 0,C 180,E1 -19580.852,E2 -19580.852} C_VEL
LIN {X 0,Y 235.263,Z 355.276,A -85,B 0,C 180,E1 -19585.417,E2 -19585.417} C_VEL
LIN {X 0,Y 235.041,Z 353.157,A -85,B 0,C 180,E1 -19590.127,E2 -19590.127} C_VEL
LIN {X 0,Y 234.939,Z 352.722,A -85,B 0,C 180,E1 -19591.403,E2 -19591.403} C_VEL
LIN {X 0,Y 234.979,Z 352.717,A -85,B 0,C 180,E1 -19595.245,E2 -19595.245} C_VEL
LIN {X 0,Y 234.991,Z 352.715,A -85,B 0,C 180,E1 -19598.967,E2 -19598.967} C_VEL
LIN {X 0,Y 235.064,Z 352.705,A -85,B 0,C 180,E1 -19603.085,E2 -19603.085} C_VEL
LIN {X 0,Y 235.115,Z 352.698,A -85,B 0,C 180,E1 -19607.921,E2 -19607.921} C_VEL
LIN {X 0,Y 235.376,Z 352.667,A -85,B 0,C 180,E1 -19611.413,E2 -19611.413} C_VEL
LIN {X 0,Y 235.403,Z 352.664,A -85,B 0,C 180,E1 -19613.14,E2 -19613.14} C_VEL
LIN {X 0,Y 235.596,Z 352.634,A -85,B 0,C 180,E1 -19618.29,E2 -19618.29} C_VEL
LIN {X 0,Y 235.595,Z 352.614,A -85,B 0,C 180,E1 -19621.708,E2 -19621.708} C_VEL
LIN {X 0,Y 235.402,Z 352.663,A -85,B 0,C 180,E1 -19626.858,E2 -19626.858} C_VEL
LIN {X 0,Y 235.237,Z 352.678,A -85,B 0,C 180,E1 -19630.326,E2 -19630.326} C_VEL
LIN {X 0,Y 235.113,Z 352.695,A -85,B 0,C 180,E1 -19635.605,E2 -19635.605} C_VEL
LIN {X 0,Y 235.006,Z 352.706,A -85,B 0,C 180,E1 -19639.205,E2 -19639.205} C_VEL
LIN {X 0,Y 234.951,Z 352.718,A -85,B 0,C 180,E1 -19642.883,E2 -19642.883} C_VEL
LIN {X 0,Y 234.967,Z 352.717,A -85,B 0,C 180,E1 -19646.656,E2 -19646.656} C_VEL
LIN {X 0,Y 234.93,Z 352.721,A -85,B 0,C 180,E1 -19650.567,E2 -19650.567} C_VEL
LIN {X 0,Y 234.958,Z 352.718,A -85,B 0,C 180,E1 -19654.632,E2 -19654.632} C_VEL
LIN {X 0,Y 234.964,Z 352.716,A -85,B 0,C 180,E1 -19658.951,E2 -19658.951} C_VEL
LIN {X 0,Y 234.963,Z 352.716,A -85,B 0,C 180,E1 -19663.467,E2 -19663.467} C_VEL
LIN {X 0,Y 234.957,Z 352.717,A -85,B 0,C 180,E1 -19666.531,E2 -19666.531} C_VEL
LIN {X 0,Y 234.952,Z 352.718,A -85,B 0,C 180,E1 -19671.086,E2 -19671.086} C_VEL
LIN {X 0,Y 234.957,Z 352.718,A -85,B 0,C 180,E1 -19675.367,E2 -19675.367} C_VEL
LIN {X 0,Y 234.93,Z 352.752,A -85,B 0,C 180,E1 -19677.979,E2 -19677.979} C_VEL
LIN {X 0,Y 235.849,Z 355.44,A -85,B 0,C 180,E1 -19678.24,E2 -19678.24} C_VEL
LIN {X 0,Y 240.368,Z 363.687,A -85,B 0,C 180,E1 -19679.308,E2 -19679.308} C_VEL
LIN {X 0,Y 245.085,Z 373.868,A -85,B 0,C 180,E1 -19680.69,E2 -19680.69} C_VEL
LIN {X 0,Y 249.82,Z 386.293,A -85,B 0,C 180,E1 -19682.509,E2 -19682.509} C_VEL
LIN {X 0,Y 253.966,Z 395.095,A -85,B 0,C 180,E1 -19684.071,E2 -19684.071} C_VEL
LIN {X 0,Y 259.756,Z 404.48,A -85,B 0,C 180,E1 -19686.056,E2 -19686.056} C_VEL
LIN {X 0,Y 267.882,Z 414.99,A -85,B 0,C 180,E1 -19688.643,E2 -19688.643} C_VEL
LIN {X 0,Y 276.518,Z 424.205,A -85,B 0,C 180,E1 -19691.215,E2 -19691.215} C_VEL
LIN {X 0,Y 285.409,Z 432.437,A -85,B 0,C 180,E1 -19693.808,E2 -19693.808} C_VEL
LIN {X 0,Y 293.215,Z 439.082,A -85,B 0,C 180,E1 -19696.132,E2 -19696.132} C_VEL
LIN {X 0,Y 299.922,Z 444.77,A -85,B 0,C 180,E1 -19698.348,E2 -19698.348} C_VEL
LIN {X 0,Y 306.241,Z 449.913,A -85,B 0,C 180,E1 -19700.681,E2 -19700.681} C_VEL
LIN {X 0,Y 309.597,Z 452.673,A -85,B 0,C 180,E1 -19702.172,E2 -19702.172} C_VEL
LIN {X 0,Y 311.899,Z 454.723,A -85,B 0,C 180,E1 -19703.531,E2 -19703.531} C_VEL
LIN {X 0,Y 313.908,Z 456.372,A -85,B 0,C 180,E1 -19704.862,E2 -19704.862} C_VEL
LIN {X 0,Y 316.701,Z 458.103,A -85,B 0,C 180,E1 -19706.959,E2 -19706.959} C_VEL
LIN {X 0,Y 318.415,Z 458.694,A -85,B 0,C 180,E1 -19708.735,E2 -19708.735} C_VEL
LIN {X 0,Y 318.983,Z 458.804,A -85,B 0,C 180,E1 -19710,E2 -19710} C_VEL
LIN {X 0,Y 318.407,Z 458.698,A -85,B 0,C 180,E1 -19711.265,E2 -19711.265} C_VEL
LIN {X 0,Y 316.694,Z 458.12,A -85,B 0,C 180,E1 -19713.018,E2 -19713.018} C_VEL
LIN {X 0,Y 313.863,Z 456.366,A -85,B 0,C 180,E1 -19715.139,E2 -19715.139} C_VEL
LIN {X 0,Y 311.403,Z 454.298,A -85,B 0,C 180,E1 -19716.776,E2 -19716.776} C_VEL
LIN {X 0,Y 308.15,Z 451.45,A -85,B 0,C 180,E1 -19718.525,E2 -19718.525} C_VEL
LIN {X 0,Y 302.571,Z 446.967,A -85,B 0,C 180,E1 -19720.709,E2 -19720.709} C_VEL
LIN {X 0,Y 296.632,Z 442.022,A -85,B 0,C 180,E1 -19722.761,E2 -19722.761} C_VEL
LIN {X 0,Y 290.574,Z 436.914,A -85,B 0,C 180,E1 -19724.659,E2 -19724.659} C_VEL
LIN {X 0,Y 282.834,Z 430.173,A -85,B 0,C 180,E1 -19726.935,E2 -19726.935} C_VEL
LIN {X 0,Y 273.584,Z 421.183,A -85,B 0,C 180,E1 -19729.656,E2 -19729.656} C_VEL
LIN {X 0,Y 265.485,Z 412.144,A -85,B 0,C 180,E1 -19732.102,E2 -19732.102} C_VEL
LIN {X 0,Y 258.639,Z 402.82,A -85,B 0,C 180,E1 -19734.32,E2 -19734.32} C_VEL
LIN {X 0,Y 253.308,Z 393.797,A -85,B 0,C 180,E1 -19736.178,E2 -19736.178} C_VEL
LIN {X 0,Y 249.137,Z 384.39,A -85,B 0,C 180,E1 -19737.79,E2 -19737.79} C_VEL
LIN {X 0,Y 243.774,Z 370.764,A -85,B 0,C 180,E1 -19739.732,E2 -19739.732} C_VEL
LIN {X 0,Y 237.869,Z 358.963,A -85,B 0,C 180,E1 -19741.311,E2 -19741.311} C_VEL
LIN {X 0,Y 236.154,Z 355.915,A -85,B 0,C 180,E1 -19741.703,E2 -19741.703} C_VEL
LIN {X 0,Y 235.05,Z 353.363,A -85,B 0,C 180,E1 -19741.979,E2 -19741.979} C_VEL
LIN {X 0,Y 234.929,Z 352.723,A -85,B 0,C 180,E1 -19742.072,E2 -19742.072} C_VEL
LIN {X 0,Y 234.954,Z 352.72,A -85,B 0,C 180,E1 -19746.137,E2 -19746.137} C_VEL
LIN {X 0,Y 234.964,Z 352.716,A -85,B 0,C 180,E1 -19748.952,E2 -19748.952} C_VEL
LIN {X 0,Y 234.957,Z 352.717,A -85,B 0,C 180,E1 -19753.469,E2 -19753.469} C_VEL
LIN {X 0,Y 234.963,Z 352.716,A -85,B 0,C 180,E1 -19756.533,E2 -19756.533} C_VEL
LIN {X 0,Y 234.952,Z 352.718,A -85,B 0,C 180,E1 -19761.087,E2 -19761.087} C_VEL
LIN {X 0,Y 234.958,Z 352.718,A -85,B 0,C 180,E1 -19765.368,E2 -19765.368} C_VEL
LIN {X 0,Y 234.967,Z 352.716,A -85,B 0,C 180,E1 -19770.158,E2 -19770.158} C_VEL
LIN {X 0,Y 234.992,Z 352.711,A -85,B 0,C 180,E1 -19773.795,E2 -19773.795} C_VEL
LIN {X 0,Y 234.996,Z 352.712,A -85,B 0,C 180,E1 -19778.97,E2 -19778.97} C_VEL
LIN {X 0,Y 235.095,Z 352.702,A -85,B 0,C 180,E1 -19783.06,E2 -19783.06} C_VEL
LIN {X 0,Y 235.146,Z 352.693,A -85,B 0,C 180,E1 -19787.925,E2 -19787.925} C_VEL
LIN {X 0,Y 235.375,Z 352.664,A -85,B 0,C 180,E1 -19791.415,E2 -19791.415} C_VEL
LIN {X 0,Y 235.402,Z 352.663,A -85,B 0,C 180,E1 -19793.142,E2 -19793.142} C_VEL
LIN {X 0,Y 235.595,Z 352.614,A -85,B 0,C 180,E1 -19798.292,E2 -19798.292} C_VEL
LIN {X 0,Y 235.596,Z 352.634,A -85,B 0,C 180,E1 -19801.71,E2 -19801.71} C_VEL
LIN {X 0,Y 235.403,Z 352.663,A -85,B 0,C 180,E1 -19806.86,E2 -19806.86} C_VEL
LIN {X 0,Y 235.238,Z 352.685,A -85,B 0,C 180,E1 -19810.327,E2 -19810.327} C_VEL
LIN {X 0,Y 235.086,Z 352.702,A -85,B 0,C 180,E1 -19815.609,E2 -19815.609} C_VEL
LIN {X 0,Y 234.991,Z 352.713,A -85,B 0,C 180,E1 -19819.208,E2 -19819.208} C_VEL
LIN {X 0,Y 234.953,Z 352.72,A -85,B 0,C 180,E1 -19822.885,E2 -19822.885} C_VEL
LIN {X 0,Y 234.969,Z 352.717,A -85,B 0,C 180,E1 -19826.658,E2 -19826.658} C_VEL
LIN {X 0,Y 234.939,Z 352.721,A -85,B 0,C 180,E1 -19828.597,E2 -19828.597} C_VEL
LIN {X 0,Y 235.152,Z 354.323,A -85,B 0,C 180,E1 -19832.546,E2 -19832.546} C_VEL
LIN {X 0,Y 235.42,Z 356.298,A -85,B 0,C 180,E1 -19836.661,E2 -19836.661} C_VEL
LIN {X 0,Y 235.796,Z 358.596,A -85,B 0,C 180,E1 -19840.975,E2 -19840.975} C_VEL
LIN {X 0,Y 235.967,Z 360.569,A -85,B 0,C 180,E1 -19844.373,E2 -19844.373} C_VEL
LIN {X 0,Y 235.839,Z 362.986,A -85,B 0,C 180,E1 -19848.16,E2 -19848.16} C_VEL
LIN {X 0,Y 235.49,Z 365.051,A -85,B 0,C 180,E1 -19851.191,E2 -19851.191} C_VEL
LIN {X 0,Y 234.753,Z 368.045,A -85,B 0,C 180,E1 -19855.332,E2 -19855.332} C_VEL
LIN {X 0,Y 234.357,Z 370.172,A -85,B 0,C 180,E1 -19858.181,E2 -19858.181} C_VEL
LIN {X 0,Y 235.314,Z 373.613,A -85,B 0,C 180,E1 -19858.497,E2 -19858.497} C_VEL
LIN {X 0,Y 239.21,Z 386.914,A -85,B 0,C 180,E1 -19860.036,E2 -19860.036} C_VEL
LIN {X 0,Y 241.272,Z 396.106,A -85,B 0,C 180,E1 -19861.209,E2 -19861.209} C_VEL
LIN {X 0,Y 241.565,Z 399.724,A -85,B 0,C 180,E1 -19861.661,E2 -19861.661} C_VEL
LIN {X 0,Y 241.048,Z 405.166,A -85,B 0,C 180,E1 -19862.273,E2 -19862.273} C_VEL
LIN {X 0,Y 237.756,Z 418.797,A -85,B 0,C 180,E1 -19864,E2 -19864} C_VEL
LIN {X 0,Y 237.235,Z 423.55,A -85,B 0,C 180,E1 -19864.849,E2 -19864.849} C_VEL
LIN {X 0,Y 237.075,Z 426.712,A -85,B 0,C 180,E1 -19865.479,E2 -19865.479} C_VEL
LIN {X 0,Y 235.031,Z 434.889,A -85,B 0,C 180,E1 -19867.125,E2 -19867.125} C_VEL
LIN {X 0,Y 232.665,Z 444.019,A -85,B 0,C 180,E1 -19869.376,E2 -19869.376} C_VEL
LIN {X 0,Y 230.64,Z 451.773,A -85,B 0,C 180,E1 -19871.8,E2 -19871.8} C_VEL
LIN {X 0,Y 229.095,Z 457.431,A -85,B 0,C 180,E1 -19873.973,E2 -19873.973} C_VEL
LIN {X 0,Y 227.567,Z 462.923,A -85,B 0,C 180,E1 -19876.607,E2 -19876.607} C_VEL
LIN {X 0,Y 226.602,Z 467.253,A -85,B 0,C 180,E1 -19879.275,E2 -19879.275} C_VEL
LIN {X 0,Y 226.146,Z 469.623,A -85,B 0,C 180,E1 -19881.061,E2 -19881.061} C_VEL
LIN {X 0,Y 225.825,Z 471.426,A -85,B 0,C 180,E1 -19882.849,E2 -19882.849} C_VEL
LIN {X 0,Y 225.595,Z 473.88,A -85,B 0,C 180,E1 -19886.428,E2 -19886.428} C_VEL
LIN {X 0,Y 225.628,Z 474.473,A -85,B 0,C 180,E1 -19888.215,E2 -19888.215} C_VEL
LIN {X 0,Y 225.714,Z 474.631,A -85,B 0,C 180,E1 -19890,E2 -19890} C_VEL
LIN {X 0,Y 225.628,Z 474.473,A -85,B 0,C 180,E1 -19891.785,E2 -19891.785} C_VEL
LIN {X 0,Y 225.592,Z 473.396,A -85,B 0,C 180,E1 -19894.49,E2 -19894.49} C_VEL
LIN {X 0,Y 225.825,Z 471.426,A -85,B 0,C 180,E1 -19897.151,E2 -19897.151} C_VEL
LIN {X 0,Y 226.349,Z 468.472,A -85,B 0,C 180,E1 -19899.833,E2 -19899.833} C_VEL
LIN {X 0,Y 227.219,Z 464.479,A -85,B 0,C 180,E1 -19902.504,E2 -19902.504} C_VEL
LIN {X 0,Y 228.537,Z 459.347,A -85,B 0,C 180,E1 -19905.153,E2 -19905.153} C_VEL
LIN {X 0,Y 230.028,Z 454.086,A -85,B 0,C 180,E1 -19907.331,E2 -19907.331} C_VEL
LIN {X 0,Y 231.777,Z 447.769,A -85,B 0,C 180,E1 -19909.484,E2 -19909.484} C_VEL
LIN {X 0,Y 233.219,Z 441.814,A -85,B 0,C 180,E1 -19911.199,E2 -19911.199} C_VEL
LIN {X 0,Y 234.986,Z 434.887,A -85,B 0,C 180,E1 -19912.88,E2 -19912.88} C_VEL
LIN {X 0,Y 237.067,Z 426.711,A -85,B 0,C 180,E1 -19914.522,E2 -19914.522} C_VEL
LIN {X 0,Y 237.191,Z 419.507,A -85,B 0,C 180,E1 -19915.915,E2 -19915.915} C_VEL
LIN {X 0,Y 236.687,Z 410.529,A -85,B 0,C 180,E1 -19917.472,E2 -19917.472} C_VEL
LIN {X 0,Y 235.255,Z 400.088,A -85,B 0,C 180,E1 -19919.094,E2 -19919.094} C_VEL
LIN {X 0,Y 233.209,Z 389.984,A -85,B 0,C 180,E1 -19920.502,E2 -19920.502} C_VEL
LIN {X 0,Y 230.366,Z 379.608,A -85,B 0,C 180,E1 -19921.822,E2 -19921.822} C_VEL
LIN {X 0,Y 228.089,Z 372.715,A -85,B 0,C 180,E1 -19922.657,E2 -19922.657} C_VEL
LIN {X 0,Y 227.451,Z 370.011,A -85,B 0,C 180,E1 -19922.923,E2 -19922.923} C_VEL
LIN {X 0,Y 228.242,Z 366.337,A -85,B 0,C 180,E1 -19928.013,E2 -19928.013} C_VEL
LIN {X 0,Y 228.817,Z 363.371,A -85,B 0,C 180,E1 -19932.51,E2 -19932.51} C_VEL
LIN {X 0,Y 228.912,Z 361.786,A -85,B 0,C 180,E1 -19935.077,E2 -19935.077} C_VEL
LIN {X 0,Y 228.846,Z 360.371,A -85,B 0,C 180,E1 -19937.496,E2 -19937.496} C_VEL
LIN {X 0,Y 228.451,Z 357.968,A -85,B 0,C 180,E1 -19942.027,E2 -19942.027} C_VEL
LIN {X 0,Y 228.207,Z 355.904,A -85,B 0,C 180,E1 -19946.334,E2 -19946.334} C_VEL
LIN {X 0,Y 227.988,Z 354.128,A -85,B 0,C 180,E1 -19950.447,E2 -19950.447} C_VEL
LIN {X 0,Y 227.943,Z 353.593,A -85,B 0,C 180,E1 -19953.397,E2 -19953.397} C_VEL
LIN {X 0,Y 227.945,Z 353.593,A -85,B 0,C 180,E1 -19958.284,E2 -19958.284} C_VEL
LIN {X 0,Y 228.009,Z 353.583,A -85,B 0,C 180,E1 -19962.847,E2 -19962.847} C_VEL
LIN {X 0,Y 228.07,Z 353.577,A -85,B 0,C 180,E1 -19967.542,E2 -19967.542} C_VEL
LIN {X 0,Y 228.306,Z 353.547,A -85,B 0,C 180,E1 -19971.145,E2 -19971.145} C_VEL
LIN {X 0,Y 228.354,Z 353.541,A -85,B 0,C 180,E1 -19972.928,E2 -19972.928} C_VEL
LIN {X 0,Y 228.555,Z 353.511,A -85,B 0,C 180,E1 -19978.237,E2 -19978.237} C_VEL
LIN {X 0,Y 228.554,Z 353.489,A -85,B 0,C 180,E1 -19981.761,E2 -19981.761} C_VEL
LIN {X 0,Y 228.353,Z 353.542,A -85,B 0,C 180,E1 -19987.07,E2 -19987.07} C_VEL
LIN {X 0,Y 228.163,Z 353.56,A -85,B 0,C 180,E1 -19990.649,E2 -19990.649} C_VEL
LIN {X 0,Y 228.064,Z 353.573,A -85,B 0,C 180,E1 -19994.271,E2 -19994.271} C_VEL
LIN {X 0,Y 228.002,Z 353.583,A -85,B 0,C 180,E1 -19997.952,E2 -19997.952} C_VEL
LIN {X 0,Y 227.915,Z 353.595,A -85,B 0,C 180,E1 -20002.32,E2 -20002.32} C_VEL
LIN {X 0,Y 227.941,Z 353.592,A -85,B 0,C 180,E1 -20006.602,E2 -20006.602} C_VEL
LIN {X 0,Y 227.907,Z 353.597,A -85,B 0,C 180,E1 -20010.295,E2 -20010.295} C_VEL
LIN {X 0,Y 227.888,Z 353.596,A -85,B 0,C 180,E1 -20013.717,E2 -20013.717} C_VEL
LIN {X 0,Y 227.869,Z 353.601,A -85,B 0,C 180,E1 -20018.085,E2 -20018.085} C_VEL
LIN {X 0,Y 227.907,Z 353.595,A -85,B 0,C 180,E1 -20022.719,E2 -20022.719} C_VEL
LIN {X 0,Y 227.895,Z 353.597,A -85,B 0,C 180,E1 -20027.741,E2 -20027.741} C_VEL
LIN {X 0,Y 227.868,Z 353.602,A -85,B 0,C 180,E1 -20031.914,E2 -20031.914} C_VEL
LIN {X 0,Y 227.888,Z 353.599,A -85,B 0,C 180,E1 -20036.372,E2 -20036.372} C_VEL
LIN {X 0,Y 227.918,Z 353.653,A -85,B 0,C 180,E1 -20036.897,E2 -20036.897} C_VEL
LIN {X 0,Y 229.065,Z 356.688,A -85,B 0,C 180,E1 -20037.234,E2 -20037.234} C_VEL
LIN {X 0,Y 233.822,Z 365.494,A -85,B 0,C 180,E1 -20038.463,E2 -20038.463} C_VEL
LIN {X 0,Y 238.542,Z 375.612,A -85,B 0,C 180,E1 -20039.943,E2 -20039.943} C_VEL
LIN {X 0,Y 242.628,Z 386.577,A -85,B 0,C 180,E1 -20041.63,E2 -20041.63} C_VEL
LIN {X 0,Y 246.155,Z 395.097,A -85,B 0,C 180,E1 -20043.152,E2 -20043.152} C_VEL
LIN {X 0,Y 250.421,Z 403.104,A -85,B 0,C 180,E1 -20044.833,E2 -20044.833} C_VEL
LIN {X 0,Y 256.974,Z 412.722,A -85,B 0,C 180,E1 -20047.188,E2 -20047.188} C_VEL
LIN {X 0,Y 265.031,Z 422.139,A -85,B 0,C 180,E1 -20049.835,E2 -20049.835} C_VEL
LIN {X 0,Y 274.818,Z 431.572,A -85,B 0,C 180,E1 -20052.849,E2 -20052.849} C_VEL
LIN {X 0,Y 283.205,Z 438.698,A -85,B 0,C 180,E1 -20055.422,E2 -20055.422} C_VEL
LIN {X 0,Y 289.379,Z 443.593,A -85,B 0,C 180,E1 -20057.375,E2 -20057.375} C_VEL
LIN {X 0,Y 296.15,Z 448.844,A -85,B 0,C 180,E1 -20059.748,E2 -20059.748} C_VEL
LIN {X 0,Y 301.73,Z 452.95,A -85,B 0,C 180,E1 -20061.966,E2 -20061.966} C_VEL
LIN {X 0,Y 304.323,Z 455.118,A -85,B 0,C 180,E1 -20063.369,E2 -20063.369} C_VEL
LIN {X 0,Y 306.412,Z 456.857,A -85,B 0,C 180,E1 -20064.736,E2 -20064.736} C_VEL
LIN {X 0,Y 308.311,Z 458.172,A -85,B 0,C 180,E1 -20066.079,E2 -20066.079} C_VEL
LIN {X 0,Y 309.993,Z 459.035,A -85,B 0,C 180,E1 -20067.401,E2 -20067.401} C_VEL
LIN {X 0,Y 311.25,Z 459.522,A -85,B 0,C 180,E1 -20068.706,E2 -20068.706} C_VEL
LIN {X 0,Y 311.909,Z 459.676,A -85,B 0,C 180,E1 -20070,E2 -20070} C_VEL
LIN {X 0,Y 311.24,Z 459.523,A -85,B 0,C 180,E1 -20071.294,E2 -20071.294} C_VEL
LIN {X 0,Y 309.623,Z 458.867,A -85,B 0,C 180,E1 -20072.896,E2 -20072.896} C_VEL
LIN {X 0,Y 308.253,Z 458.176,A -85,B 0,C 180,E1 -20073.922,E2 -20073.922} C_VEL
LIN {X 0,Y 306.379,Z 456.858,A -85,B 0,C 180,E1 -20075.265,E2 -20075.265} C_VEL
LIN {X 0,Y 303.104,Z 454.069,A -85,B 0,C 180,E1 -20077.326,E2 -20077.326} C_VEL
LIN {X 0,Y 301.708,Z 452.951,A -85,B 0,C 180,E1 -20078.034,E2 -20078.034} C_VEL
LIN {X 0,Y 296.151,Z 448.844,A -85,B 0,C 180,E1 -20080.252,E2 -20080.252} C_VEL
LIN {X 0,Y 289.384,Z 443.593,A -85,B 0,C 180,E1 -20082.625,E2 -20082.625} C_VEL
LIN {X 0,Y 281.912,Z 437.641,A -85,B 0,C 180,E1 -20084.982,E2 -20084.982} C_VEL
LIN {X 0,Y 272.963,Z 429.903,A -85,B 0,C 180,E1 -20087.707,E2 -20087.707} C_VEL
LIN {X 0,Y 264.313,Z 421.325,A -85,B 0,C 180,E1 -20090.402,E2 -20090.402} C_VEL
LIN {X 0,Y 255.544,Z 410.891,A -85,B 0,C 180,E1 -20093.291,E2 -20093.291} C_VEL
LIN {X 0,Y 249.353,Z 401.188,A -85,B 0,C 180,E1 -20095.591,E2 -20095.591} C_VEL
LIN {X 0,Y 245.109,Z 392.679,A -85,B 0,C 180,E1 -20097.307,E2 -20097.307} C_VEL
LIN {X 0,Y 241.163,Z 382.349,A -85,B 0,C 180,E1 -20099.044,E2 -20099.044} C_VEL
LIN {X 0,Y 236.429,Z 370.767,A -85,B 0,C 180,E1 -20100.769,E2 -20100.769} C_VEL
LIN {X 0,Y 230.686,Z 359.595,A -85,B 0,C 180,E1 -20102.382,E2 -20102.382} C_VEL
LIN {X 0,Y 229.189,Z 356.834,A -85,B 0,C 180,E1 -20102.754,E2 -20102.754} C_VEL
LIN {X 0,Y 227.99,Z 354.111,A -85,B 0,C 180,E1 -20103.071,E2 -20103.071} C_VEL
LIN {X 0,Y 227.901,Z 353.597,A -85,B 0,C 180,E1 -20103.156,E2 -20103.156} C_VEL
LIN {X 0,Y 227.905,Z 353.596,A -85,B 0,C 180,E1 -20106.702,E2 -20106.702} C_VEL
LIN {X 0,Y 227.875,Z 353.599,A -85,B 0,C 180,E1 -20110.366,E2 -20110.366} C_VEL
LIN {X 0,Y 227.899,Z 353.595,A -85,B 0,C 180,E1 -20112.722,E2 -20112.722} C_VEL
LIN {X 0,Y 227.907,Z 353.596,A -85,B 0,C 180,E1 -20117.739,E2 -20117.739} C_VEL
LIN {X 0,Y 227.869,Z 353.601,A -85,B 0,C 180,E1 -20121.915,E2 -20121.915} C_VEL
LIN {X 0,Y 227.888,Z 353.596,A -85,B 0,C 180,E1 -20126.374,E2 -20126.374} C_VEL
LIN {X 0,Y 227.917,Z 353.594,A -85,B 0,C 180,E1 -20130.439,E2 -20130.439} C_VEL
LIN {X 0,Y 227.923,Z 353.589,A -85,B 0,C 180,E1 -20134.426,E2 -20134.426} C_VEL
LIN {X 0,Y 227.946,Z 353.589,A -85,B 0,C 180,E1 -20138.287,E2 -20138.287} C_VEL
LIN {X 0,Y 228.034,Z 353.58,A -85,B 0,C 180,E1 -20142.827,E2 -20142.827} C_VEL
LIN {X 0,Y 228.093,Z 353.573,A -85,B 0,C 180,E1 -20147.545,E2 -20147.545} C_VEL
LIN {X 0,Y 228.305,Z 353.543,A -85,B 0,C 180,E1 -20151.147,E2 -20151.147} C_VEL
LIN {X 0,Y 228.353,Z 353.542,A -85,B 0,C 180,E1 -20152.93,E2 -20152.93} C_VEL
LIN {X 0,Y 228.554,Z 353.489,A -85,B 0,C 180,E1 -20158.239,E2 -20158.239} C_VEL
LIN {X 0,Y 228.555,Z 353.511,A -85,B 0,C 180,E1 -20161.763,E2 -20161.763} C_VEL
LIN {X 0,Y 228.354,Z 353.541,A -85,B 0,C 180,E1 -20167.072,E2 -20167.072} C_VEL
LIN {X 0,Y 228.159,Z 353.567,A -85,B 0,C 180,E1 -20170.652,E2 -20170.652} C_VEL
LIN {X 0,Y 228.049,Z 353.582,A -85,B 0,C 180,E1 -20174.274,E2 -20174.274} C_VEL
LIN {X 0,Y 227.969,Z 353.59,A -85,B 0,C 180,E1 -20177.957,E2 -20177.957} C_VEL
LIN {X 0,Y 227.917,Z 353.597,A -85,B 0,C 180,E1 -20182.321,E2 -20182.321} C_VEL
LIN {X 0,Y 227.943,Z 353.593,A -85,B 0,C 180,E1 -20186.603,E2 -20186.603} C_VEL
LIN {X 0,Y 227.987,Z 354.123,A -85,B 0,C 180,E1 -20189.553,E2 -20189.553} C_VEL
LIN {X 0,Y 228.202,Z 355.934,A -85,B 0,C 180,E1 -20193.745,E2 -20193.745} C_VEL
LIN {X 0,Y 228.452,Z 357.978,A -85,B 0,C 180,E1 -20197.973,E2 -20197.973} C_VEL
LIN {X 0,Y 228.672,Z 359.124,A -85,B 0,C 180,E1 -20200.198,E2 -20200.198} C_VEL
LIN {X 0,Y 228.844,Z 360.405,A -85,B 0,C 180,E1 -20202.519,E2 -20202.519} C_VEL
LIN {X 0,Y 228.914,Z 361.895,A -85,B 0,C 180,E1 -20205.079,E2 -20205.079} C_VEL
LIN {X 0,Y 228.817,Z 363.379,A -85,B 0,C 180,E1 -20207.49,E2 -20207.49} C_VEL
LIN {X 0,Y 228.497,Z 365.204,A -85,B 0,C 180,E1 -20210.26,E2 -20210.26} C_VEL
LIN {X 0,Y 227.866,Z 367.862,A -85,B 0,C 180,E1 -20214.126,E2 -20214.126} C_VEL
LIN {X 0,Y 227.443,Z 369.974,A -85,B 0,C 180,E1 -20217.08,E2 -20217.08} C_VEL
LIN {X 0,Y 228.374,Z 373.336,A -85,B 0,C 180,E1 -20217.421,E2 -20217.421} C_VEL
LIN {X 0,Y 231.98,Z 385.201,A -85,B 0,C 180,E1 -20218.856,E2 -20218.856} C_VEL
LIN {X 0,Y 234.553,Z 396.172,A -85,B 0,C 180,E1 -20220.337,E2 -20220.337} C_VEL
LIN {X 0,Y 236.142,Z 405.948,A -85,B 0,C 180,E1 -20221.789,E2 -20221.789} C_VEL
LIN {X 0,Y 237.01,Z 414.894,A -85,B 0,C 180,E1 -20223.261,E2 -20223.261} C_VEL
LIN {X 0,Y 237.235,Z 423.55,A -85,B 0,C 180,E1 -20224.849,E2 -20224.849} C_VEL
LIN {X 0,Y 236.634,Z 426.155,A -85,B 0,C 180,E1 -20225.315,E2 -20225.315} C_VEL
LIN {X 0,Y 234.454,Z 429.672,A -85,B 0,C 180,E1 -20225.818,E2 -20225.818} C_VEL
LIN {X 0,Y 228.781,Z 436.286,A -85,B 0,C 180,E1 -20226.844,E2 -20226.844} C_VEL
LIN {X 0,Y 227.292,Z 439.085,A -85,B 0,C 180,E1 -20227.476,E2 -20227.476} C_VEL
LIN {X 0,Y 225.351,Z 446.409,A -85,B 0,C 180,E1 -20229.535,E2 -20229.535} C_VEL
LIN {X 0,Y 223.516,Z 452.732,A -85,B 0,C 180,E1 -20231.674,E2 -20231.674} C_VEL
LIN {X 0,Y 222.263,Z 457.235,A -85,B 0,C 180,E1 -20233.466,E2 -20233.466} C_VEL
LIN {X 0,Y 220.629,Z 462.726,A -85,B 0,C 180,E1 -20236.178,E2 -20236.178} C_VEL
LIN {X 0,Y 219.61,Z 467.057,A -85,B 0,C 180,E1 -20238.93,E2 -20238.93} C_VEL
LIN {X 0,Y 219.098,Z 469.426,A -85,B 0,C 180,E1 -20240.771,E2 -20240.771} C_VEL
LIN {X 0,Y 218.763,Z 471.229,A -85,B 0,C 180,E1 -20242.617,E2 -20242.617} C_VEL
LIN {X 0,Y 218.501,Z 473.684,A -85,B 0,C 180,E1 -20246.312,E2 -20246.312} C_VEL
LIN {X 0,Y 218.528,Z 474.277,A -85,B 0,C 180,E1 -20248.157,E2 -20248.157} C_VEL
LIN {X 0,Y 218.629,Z 474.435,A -85,B 0,C 180,E1 -20250,E2 -20250} C_VEL
LIN {X 0,Y 218.527,Z 474.277,A -85,B 0,C 180,E1 -20251.843,E2 -20251.843} C_VEL
LIN {X 0,Y 218.488,Z 473.41,A -85,B 0,C 180,E1 -20254.307,E2 -20254.307} C_VEL
LIN {X 0,Y 218.763,Z 471.229,A -85,B 0,C 180,E1 -20257.383,E2 -20257.383} C_VEL
LIN {X 0,Y 219.334,Z 468.275,A -85,B 0,C 180,E1 -20260.15,E2 -20260.15} C_VEL
LIN {X 0,Y 220.239,Z 464.281,A -85,B 0,C 180,E1 -20262.907,E2 -20262.907} C_VEL
LIN {X 0,Y 221.674,Z 459.151,A -85,B 0,C 180,E1 -20265.634,E2 -20265.634} C_VEL
LIN {X 0,Y 223.216,Z 453.889,A -85,B 0,C 180,E1 -20267.877,E2 -20267.877} C_VEL
LIN {X 0,Y 225.053,Z 447.572,A -85,B 0,C 180,E1 -20270.091,E2 -20270.091} C_VEL
LIN {X 0,Y 227.012,Z 439.989,A -85,B 0,C 180,E1 -20272.287,E2 -20272.287} C_VEL
LIN {X 0,Y 229.508,Z 430.854,A -85,B 0,C 180,E1 -20274.418,E2 -20274.418} C_VEL
LIN {X 0,Y 230.487,Z 426.511,A -85,B 0,C 180,E1 -20275.27,E2 -20275.27} C_VEL
LIN {X 0,Y 230.475,Z 417.94,A -85,B 0,C 180,E1 -20276.974,E2 -20276.974} C_VEL
LIN {X 0,Y 229.851,Z 409.153,A -85,B 0,C 180,E1 -20278.538,E2 -20278.538} C_VEL
LIN {X 0,Y 228.456,Z 399.519,A -85,B 0,C 180,E1 -20280.091,E2 -20280.091} C_VEL
LIN {X 0,Y 226.553,Z 390.239,A -85,B 0,C 180,E1 -20281.451,E2 -20281.451} C_VEL
LIN {X 0,Y 223.755,Z 379.951,A -85,B 0,C 180,E1 -20282.836,E2 -20282.836} C_VEL
LIN {X 0,Y 221.385,Z 372.996,A -85,B 0,C 180,E1 -20283.749,E2 -20283.749} C_VEL
LIN {X 0,Y 220.532,Z 369.825,A -85,B 0,C 180,E1 -20284.096,E2 -20284.096} C_VEL
LIN {X 0,Y 221.046,Z 367.519,A -85,B 0,C 180,E1 -20287.357,E2 -20287.357} C_VEL
LIN {X 0,Y 221.501,Z 365.537,A -85,B 0,C 180,E1 -20290.402,E2 -20290.402} C_VEL
LIN {X 0,Y 221.817,Z 363.195,A -85,B 0,C 180,E1 -20294.19,E2 -20294.19} C_VEL
LIN {X 0,Y 221.716,Z 360.88,A -85,B 0,C 180,E1 -20298.266,E2 -20298.266} C_VEL
LIN {X 0,Y 221.371,Z 358.54,A -85,B 0,C 180,E1 -20302.899,E2 -20302.899} C_VEL
LIN {X 0,Y 221.085,Z 356.533,A -85,B 0,C 180,E1 -20307.288,E2 -20307.288} C_VEL
LIN {X 0,Y 220.866,Z 354.833,A -85,B 0,C 180,E1 -20311.49,E2 -20311.49} C_VEL
LIN {X 0,Y 220.895,Z 354.471,A -85,B 0,C 180,E1 -20313.548,E2 -20313.548} C_VEL
LIN {X 0,Y 220.865,Z 354.476,A -85,B 0,C 180,E1 -20317.551,E2 -20317.551} C_VEL
LIN {X 0,Y 220.963,Z 354.461,A -85,B 0,C 180,E1 -20322.589,E2 -20322.589} C_VEL
LIN {X 0,Y 221.007,Z 354.456,A -85,B 0,C 180,E1 -20327.137,E2 -20327.137} C_VEL
LIN {X 0,Y 221.237,Z 354.427,A -85,B 0,C 180,E1 -20330.86,E2 -20330.86} C_VEL
LIN {X 0,Y 221.289,Z 354.42,A -85,B 0,C 180,E1 -20332.701,E2 -20332.701} C_VEL
LIN {X 0,Y 221.513,Z 354.388,A -85,B 0,C 180,E1 -20338.181,E2 -20338.181} C_VEL
LIN {X 0,Y 221.512,Z 354.365,A -85,B 0,C 180,E1 -20341.817,E2 -20341.817} C_VEL
LIN {X 0,Y 221.288,Z 354.42,A -85,B 0,C 180,E1 -20347.297,E2 -20347.297} C_VEL
LIN {X 0,Y 221.112,Z 354.441,A -85,B 0,C 180,E1 -20350.993,E2 -20350.993} C_VEL
LIN {X 0,Y 221.015,Z 354.454,A -85,B 0,C 180,E1 -20356.629,E2 -20356.629} C_VEL
LIN {X 0,Y 220.883,Z 354.465,A -85,B 0,C 180,E1 -20360.486,E2 -20360.486} C_VEL
LIN {X 0,Y 220.86,Z 354.469,A -85,B 0,C 180,E1 -20364.435,E2 -20364.435} C_VEL
LIN {X 0,Y 220.835,Z 354.477,A -85,B 0,C 180,E1 -20368.513,E2 -20368.513} C_VEL
LIN {X 0,Y 220.822,Z 354.477,A -85,B 0,C 180,E1 -20372.754,E2 -20372.754} C_VEL
LIN {X 0,Y 220.836,Z 354.476,A -85,B 0,C 180,E1 -20377.287,E2 -20377.287} C_VEL
LIN {X 0,Y 220.851,Z 354.476,A -85,B 0,C 180,E1 -20381.932,E2 -20381.932} C_VEL
LIN {X 0,Y 220.859,Z 354.472,A -85,B 0,C 180,E1 -20387.043,E2 -20387.043} C_VEL
LIN {X 0,Y 220.849,Z 354.476,A -85,B 0,C 180,E1 -20390.472,E2 -20390.472} C_VEL
LIN {X 0,Y 220.813,Z 354.48,A -85,B 0,C 180,E1 -20395.047,E2 -20395.047} C_VEL
LIN {X 0,Y 220.852,Z 354.549,A -85,B 0,C 180,E1 -20395.727,E2 -20395.727} C_VEL
LIN {X 0,Y 221.809,Z 357.29,A -85,B 0,C 180,E1 -20396.038,E2 -20396.038} C_VEL
LIN {X 0,Y 223.253,Z 359.579,A -85,B 0,C 180,E1 -20396.406,E2 -20396.406} C_VEL
LIN {X 0,Y 228.383,Z 369.49,A -85,B 0,C 180,E1 -20397.908,E2 -20397.908} C_VEL
LIN {X 0,Y 232.669,Z 378.917,A -85,B 0,C 180,E1 -20399.411,E2 -20399.411} C_VEL
LIN {X 0,Y 236.655,Z 390.026,A -85,B 0,C 180,E1 -20401.247,E2 -20401.247} C_VEL
LIN {X 0,Y 240.24,Z 398.95,A -85,B 0,C 180,E1 -20402.975,E2 -20402.975} C_VEL
LIN {X 0,Y 244.573,Z 407.125,A -85,B 0,C 180,E1 -20404.843,E2 -20404.843} C_VEL
LIN {X 0,Y 251.197,Z 416.743,A -85,B 0,C 180,E1 -20407.407,E2 -20407.407} C_VEL
LIN {X 0,Y 259.449,Z 426.103,A -85,B 0,C 180,E1 -20410.269,E2 -20410.269} C_VEL
LIN {X 0,Y 268.821,Z 434.721,A -85,B 0,C 180,E1 -20413.287,E2 -20413.287} C_VEL
LIN {X 0,Y 275.829,Z 440.426,A -85,B 0,C 180,E1 -20415.514,E2 -20415.514} C_VEL
LIN {X 0,Y 281.099,Z 444.309,A -85,B 0,C 180,E1 -20417.176,E2 -20417.176} C_VEL
LIN {X 0,Y 288.114,Z 449.416,A -85,B 0,C 180,E1 -20419.62,E2 -20419.62} C_VEL
LIN {X 0,Y 293.53,Z 453.177,A -85,B 0,C 180,E1 -20421.74,E2 -20421.74} C_VEL
LIN {X 0,Y 296.633,Z 455.332,A -85,B 0,C 180,E1 -20423.197,E2 -20423.197} C_VEL
LIN {X 0,Y 298.845,Z 457.068,A -85,B 0,C 180,E1 -20424.602,E2 -20424.602} C_VEL
LIN {X 0,Y 300.861,Z 458.398,A -85,B 0,C 180,E1 -20425.981,E2 -20425.981} C_VEL
LIN {X 0,Y 302.683,Z 459.339,A -85,B 0,C 180,E1 -20427.338,E2 -20427.338} C_VEL
LIN {X 0,Y 304.039,Z 459.899,A -85,B 0,C 180,E1 -20428.675,E2 -20428.675} C_VEL
LIN {X 0,Y 304.805,Z 460.082,A -85,B 0,C 180,E1 -20430,E2 -20430} C_VEL
LIN {X 0,Y 304.006,Z 459.9,A -85,B 0,C 180,E1 -20431.325,E2 -20431.325} C_VEL
LIN {X 0,Y 302.543,Z 459.299,A -85,B 0,C 180,E1 -20432.73,E2 -20432.73} C_VEL
LIN {X 0,Y 300.786,Z 458.399,A -85,B 0,C 180,E1 -20434.02,E2 -20434.02} C_VEL
LIN {X 0,Y 298.816,Z 457.069,A -85,B 0,C 180,E1 -20435.398,E2 -20435.398} C_VEL
LIN {X 0,Y 296.632,Z 455.332,A -85,B 0,C 180,E1 -20436.803,E2 -20436.803} C_VEL
LIN {X 0,Y 293.501,Z 453.178,A -85,B 0,C 180,E1 -20438.26,E2 -20438.26} C_VEL
LIN {X 0,Y 288.12,Z 449.406,A -85,B 0,C 180,E1 -20440.384,E2 -20440.384} C_VEL
LIN {X 0,Y 281.095,Z 444.319,A -85,B 0,C 180,E1 -20442.82,E2 -20442.82} C_VEL
LIN {X 0,Y 272.19,Z 437.528,A -85,B 0,C 180,E1 -20445.648,E2 -20445.648} C_VEL
LIN {X 0,Y 262.51,Z 429.041,A -85,B 0,C 180,E1 -20448.739,E2 -20448.739} C_VEL
LIN {X 0,Y 254.867,Z 421.17,A -85,B 0,C 180,E1 -20451.289,E2 -20451.289} C_VEL
LIN {X 0,Y 248.091,Z 412.575,A -85,B 0,C 180,E1 -20453.758,E2 -20453.758} C_VEL
LIN {X 0,Y 242.488,Z 403.382,A -85,B 0,C 180,E1 -20456.045,E2 -20456.045} C_VEL
LIN {X 0,Y 238.486,Z 394.788,A -85,B 0,C 180,E1 -20457.864,E2 -20457.864} C_VEL
LIN {X 0,Y 234.213,Z 382.914,A -85,B 0,C 180,E1 -20459.954,E2 -20459.954} C_VEL
LIN {X 0,Y 229.118,Z 370.934,A -85,B 0,C 180,E1 -20461.868,E2 -20461.868} C_VEL
LIN {X 0,Y 222.769,Z 358.523,A -85,B 0,C 180,E1 -20463.754,E2 -20463.754} C_VEL
LIN {X 0,Y 221.206,Z 356.064,A -85,B 0,C 180,E1 -20464.142,E2 -20464.142} C_VEL
LIN {X 0,Y 220.821,Z 354.48,A -85,B 0,C 180,E1 -20464.347,E2 -20464.347} C_VEL
LIN {X 0,Y 220.835,Z 354.477,A -85,B 0,C 180,E1 -20467.288,E2 -20467.288} C_VEL
LIN {X 0,Y 220.84,Z 354.477,A -85,B 0,C 180,E1 -20471.936,E2 -20471.936} C_VEL
LIN {X 0,Y 220.865,Z 354.472,A -85,B 0,C 180,E1 -20477.043,E2 -20477.043} C_VEL
LIN {X 0,Y 220.854,Z 354.474,A -85,B 0,C 180,E1 -20480.475,E2 -20480.475} C_VEL
LIN {X 0,Y 220.813,Z 354.479,A -85,B 0,C 180,E1 -20485.049,E2 -20485.049} C_VEL
LIN {X 0,Y 220.866,Z 354.473,A -85,B 0,C 180,E1 -20489.396,E2 -20489.396} C_VEL
LIN {X 0,Y 220.893,Z 354.468,A -85,B 0,C 180,E1 -20493.55,E2 -20493.55} C_VEL
LIN {X 0,Y 220.864,Z 354.474,A -85,B 0,C 180,E1 -20497.553,E2 -20497.553} C_VEL
LIN {X 0,Y 220.983,Z 354.458,A -85,B 0,C 180,E1 -20502.572,E2 -20502.572} C_VEL
LIN {X 0,Y 221.025,Z 354.453,A -85,B 0,C 180,E1 -20507.14,E2 -20507.14} C_VEL
LIN {X 0,Y 221.235,Z 354.421,A -85,B 0,C 180,E1 -20510.862,E2 -20510.862} C_VEL
LIN {X 0,Y 221.288,Z 354.42,A -85,B 0,C 180,E1 -20512.703,E2 -20512.703} C_VEL
LIN {X 0,Y 221.512,Z 354.365,A -85,B 0,C 180,E1 -20518.183,E2 -20518.183} C_VEL
LIN {X 0,Y 221.513,Z 354.388,A -85,B 0,C 180,E1 -20521.819,E2 -20521.819} C_VEL
LIN {X 0,Y 221.289,Z 354.42,A -85,B 0,C 180,E1 -20527.299,E2 -20527.299} C_VEL
LIN {X 0,Y 221.106,Z 354.445,A -85,B 0,C 180,E1 -20530.995,E2 -20530.995} C_VEL
LIN {X 0,Y 220.992,Z 354.46,A -85,B 0,C 180,E1 -20536.633,E2 -20536.633} C_VEL
LIN {X 0,Y 220.877,Z 354.473,A -85,B 0,C 180,E1 -20540.489,E2 -20540.489} C_VEL
LIN {X 0,Y 220.863,Z 354.476,A -85,B 0,C 180,E1 -20544.437,E2 -20544.437} C_VEL
LIN {X 0,Y 220.885,Z 354.472,A -85,B 0,C 180,E1 -20547.015,E2 -20547.015} C_VEL
LIN {X 0,Y 221.011,Z 355.752,A -85,B 0,C 180,E1 -20550.843,E2 -20550.843} C_VEL
LIN {X 0,Y 221.234,Z 357.492,A -85,B 0,C 180,E1 -20554.878,E2 -20554.878} C_VEL
LIN {X 0,Y 221.557,Z 359.678,A -85,B 0,C 180,E1 -20559.378,E2 -20559.378} C_VEL
LIN {X 0,Y 221.782,Z 361.732,A -85,B 0,C 180,E1 -20563.211,E2 -20563.211} C_VEL
LIN {X 0,Y 221.753,Z 363.796,A -85,B 0,C 180,E1 -20566.799,E2 -20566.799} C_VEL
LIN {X 0,Y 221.36,Z 366.184,A -85,B 0,C 180,E1 -20570.582,E2 -20570.582} C_VEL
LIN {X 0,Y 221.034,Z 367.672,A -85,B 0,C 180,E1 -20572.834,E2 -20572.834} C_VEL
LIN {X 0,Y 220.524,Z 369.783,A -85,B 0,C 180,E1 -20575.906,E2 -20575.906} C_VEL
LIN {X 0,Y 221.477,Z 373.139,A -85,B 0,C 180,E1 -20576.275,E2 -20576.275} C_VEL
LIN {X 0,Y 225.281,Z 385.217,A -85,B 0,C 180,E1 -20577.844,E2 -20577.844} C_VEL
LIN {X 0,Y 227.781,Z 395.661,A -85,B 0,C 180,E1 -20579.325,E2 -20579.325} C_VEL
LIN {X 0,Y 229.475,Z 406.016,A -85,B 0,C 180,E1 -20580.934,E2 -20580.934} C_VEL
LIN {X 0,Y 230.367,Z 415.209,A -85,B 0,C 180,E1 -20582.52,E2 -20582.52} C_VEL
LIN {X 0,Y 230.542,Z 424.227,A -85,B 0,C 180,E1 -20584.253,E2 -20584.253} C_VEL
LIN {X 0,Y 230.357,Z 427.65,A -85,B 0,C 180,E1 -20584.956,E2 -20584.956} C_VEL
LIN {X 0,Y 227.505,Z 438.363,A -85,B 0,C 180,E1 -20587.285,E2 -20587.285} C_VEL
LIN {X 0,Y 227.292,Z 439.085,A -85,B 0,C 180,E1 -20587.476,E2 -20587.476} C_VEL
LIN {X 0,Y 225.55,Z 443.173,A -85,B 0,C 180,E1 -20588.498,E2 -20588.498} C_VEL
LIN {X 0,Y 221.132,Z 449.206,A -85,B 0,C 180,E1 -20590.148,E2 -20590.148} C_VEL
LIN {X 0,Y 216.804,Z 454.739,A -85,B 0,C 180,E1 -20591.975,E2 -20591.975} C_VEL
LIN {X 0,Y 215.226,Z 457.725,A -85,B 0,C 180,E1 -20593.259,E2 -20593.259} C_VEL
LIN {X 0,Y 213.714,Z 462.529,A -85,B 0,C 180,E1 -20595.721,E2 -20595.721} C_VEL
LIN {X 0,Y 212.612,Z 466.86,A -85,B 0,C 180,E1 -20598.561,E2 -20598.561} C_VEL
LIN {X 0,Y 212.072,Z 469.23,A -85,B 0,C 180,E1 -20600.462,E2 -20600.462} C_VEL
LIN {X 0,Y 211.691,Z 471.033,A -85,B 0,C 180,E1 -20602.369,E2 -20602.369} C_VEL
LIN {X 0,Y 211.42,Z 473.488,A -85,B 0,C 180,E1 -20606.188,E2 -20606.188} C_VEL
LIN {X 0,Y 211.43,Z 474.081,A -85,B 0,C 180,E1 -20608.095,E2 -20608.095} C_VEL
LIN {X 0,Y 211.545,Z 474.24,A -85,B 0,C 180,E1 -20610,E2 -20610} C_VEL
LIN {X 0,Y 211.429,Z 474.081,A -85,B 0,C 180,E1 -20611.905,E2 -20611.905} C_VEL
LIN {X 0,Y 211.396,Z 473.372,A -85,B 0,C 180,E1 -20614.145,E2 -20614.145} C_VEL
LIN {X 0,Y 211.691,Z 471.033,A -85,B 0,C 180,E1 -20617.631,E2 -20617.631} C_VEL
LIN {X 0,Y 212.337,Z 468.079,A -85,B 0,C 180,E1 -20620.489,E2 -20620.489} C_VEL
LIN {X 0,Y 213.275,Z 464.084,A -85,B 0,C 180,E1 -20623.336,E2 -20623.336} C_VEL
LIN {X 0,Y 214.833,Z 458.954,A -85,B 0,C 180,E1 -20626.145,E2 -20626.145} C_VEL
LIN {X 0,Y 216.413,Z 453.691,A -85,B 0,C 180,E1 -20628.459,E2 -20628.459} C_VEL
LIN {X 0,Y 218.366,Z 447.375,A -85,B 0,C 180,E1 -20630.734,E2 -20630.734} C_VEL
LIN {X 0,Y 219.963,Z 441.42,A -85,B 0,C 180,E1 -20632.545,E2 -20632.545} C_VEL
LIN {X 0,Y 221.939,Z 434.495,A -85,B 0,C 180,E1 -20634.309,E2 -20634.309} C_VEL
LIN {X 0,Y 223.803,Z 427.45,A -85,B 0,C 180,E1 -20635.83,E2 -20635.83} C_VEL
LIN {X 0,Y 223.897,Z 419.334,A -85,B 0,C 180,E1 -20637.536,E2 -20637.536} C_VEL
LIN {X 0,Y 223.342,Z 410.705,A -85,B 0,C 180,E1 -20639.173,E2 -20639.173} C_VEL
LIN {X 0,Y 222.015,Z 400.782,A -85,B 0,C 180,E1 -20640.868,E2 -20640.868} C_VEL
LIN {X 0,Y 220.259,Z 391.85,A -85,B 0,C 180,E1 -20642.268,E2 -20642.268} C_VEL
LIN {X 0,Y 217.116,Z 380.21,A -85,B 0,C 180,E1 -20643.935,E2 -20643.935} C_VEL
LIN {X 0,Y 214.47,Z 372.789,A -85,B 0,C 180,E1 -20644.991,E2 -20644.991} C_VEL
LIN {X 0,Y 213.623,Z 369.658,A -85,B 0,C 180,E1 -20645.33,E2 -20645.33} C_VEL
LIN {X 0,Y 214.149,Z 367.472,A -85,B 0,C 180,E1 -20648.575,E2 -20648.575} C_VEL
LIN {X 0,Y 214.49,Z 365.891,A -85,B 0,C 180,E1 -20651.094,E2 -20651.094} C_VEL
LIN {X 0,Y 214.741,Z 364.192,A -85,B 0,C 180,E1 -20653.943,E2 -20653.943} C_VEL
LIN {X 0,Y 214.737,Z 362.71,A -85,B 0,C 180,E1 -20656.582,E2 -20656.582} C_VEL
LIN {X 0,Y 214.627,Z 361.39,A -85,B 0,C 180,E1 -20659.086,E2 -20659.086} C_VEL
LIN {X 0,Y 214.27,Z 359.116,A -85,B 0,C 180,E1 -20663.814,E2 -20663.814} C_VEL
LIN {X 0,Y 213.998,Z 357.036,A -85,B 0,C 180,E1 -20668.635,E2 -20668.635} C_VEL
LIN {X 0,Y 213.846,Z 355.518,A -85,B 0,C 180,E1 -20672.605,E2 -20672.605} C_VEL
LIN {X 0,Y 213.82,Z 355.353,A -85,B 0,C 180,E1 -20676.973,E2 -20676.973} C_VEL
LIN {X 0,Y 213.922,Z 355.338,A -85,B 0,C 180,E1 -20682.801,E2 -20682.801} C_VEL
LIN {X 0,Y 213.946,Z 355.335,A -85,B 0,C 180,E1 -20686.705,E2 -20686.705} C_VEL
LIN {X 0,Y 214.168,Z 355.307,A -85,B 0,C 180,E1 -20690.555,E2 -20690.555} C_VEL
LIN {X 0,Y 214.227,Z 355.299,A -85,B 0,C 180,E1 -20692.459,E2 -20692.459} C_VEL
LIN {X 0,Y 214.446,Z 355.269,A -85,B 0,C 180,E1 -20698.121,E2 -20698.121} C_VEL
LIN {X 0,Y 214.546,Z 355.244,A -85,B 0,C 180,E1 -20699.999,E2 -20699.999} C_VEL
LIN {X 0,Y 214.445,Z 355.244,A -85,B 0,C 180,E1 -20701.877,E2 -20701.877} C_VEL
LIN {X 0,Y 214.226,Z 355.299,A -85,B 0,C 180,E1 -20707.539,E2 -20707.539} C_VEL
LIN {X 0,Y 214.044,Z 355.323,A -85,B 0,C 180,E1 -20711.361,E2 -20711.361} C_VEL
LIN {X 0,Y 213.933,Z 355.332,A -85,B 0,C 180,E1 -20715.236,E2 -20715.236} C_VEL
LIN {X 0,Y 213.834,Z 355.342,A -85,B 0,C 180,E1 -20719.187,E2 -20719.187} C_VEL
LIN {X 0,Y 213.809,Z 355.35,A -85,B 0,C 180,E1 -20723.23,E2 -20723.23} C_VEL
LIN {X 0,Y 213.827,Z 355.349,A -85,B 0,C 180,E1 -20727.449,E2 -20727.449} C_VEL
LIN {X 0,Y 213.777,Z 355.355,A -85,B 0,C 180,E1 -20731.735,E2 -20731.735} C_VEL
LIN {X 0,Y 213.752,Z 355.359,A -85,B 0,C 180,E1 -20736.285,E2 -20736.285} C_VEL
LIN {X 0,Y 213.791,Z 355.354,A -85,B 0,C 180,E1 -20741.105,E2 -20741.105} C_VEL
LIN {X 0,Y 213.806,Z 355.352,A -85,B 0,C 180,E1 -20743.684,E2 -20743.684} C_VEL
LIN {X 0,Y 213.809,Z 355.352,A -85,B 0,C 180,E1 -20746.348,E2 -20746.348} C_VEL
LIN {X 0,Y 213.776,Z 355.356,A -85,B 0,C 180,E1 -20751.345,E2 -20751.345} C_VEL
LIN {X 0,Y 213.766,Z 355.378,A -85,B 0,C 180,E1 -20754.454,E2 -20754.454} C_VEL
LIN {X 0,Y 214.741,Z 358.176,A -85,B 0,C 180,E1 -20754.793,E2 -20754.793} C_VEL
LIN {X 0,Y 216.26,Z 360.56,A -85,B 0,C 180,E1 -20755.205,E2 -20755.205} C_VEL
LIN {X 0,Y 221.17,Z 369.752,A -85,B 0,C 180,E1 -20756.732,E2 -20756.732} C_VEL
LIN {X 0,Y 226.295,Z 381.076,A -85,B 0,C 180,E1 -20758.654,E2 -20758.654} C_VEL
LIN {X 0,Y 230.073,Z 391.628,A -85,B 0,C 180,E1 -20760.526,E2 -20760.526} C_VEL
LIN {X 0,Y 233.894,Z 401.887,A -85,B 0,C 180,E1 -20762.619,E2 -20762.619} C_VEL
LIN {X 0,Y 238.957,Z 411.512,A -85,B 0,C 180,E1 -20765.005,E2 -20765.005} C_VEL
LIN {X 0,Y 245.1,Z 420.301,A -85,B 0,C 180,E1 -20767.549,E2 -20767.549} C_VEL
LIN {X 0,Y 253.349,Z 429.423,A -85,B 0,C 180,E1 -20770.588,E2 -20770.588} C_VEL
LIN {X 0,Y 262.022,Z 437.121,A -85,B 0,C 180,E1 -20773.51,E2 -20773.51} C_VEL
LIN {X 0,Y 271.209,Z 444.108,A -85,B 0,C 180,E1 -20776.513,E2 -20776.513} C_VEL
LIN {X 0,Y 276.485,Z 447.706,A -85,B 0,C 180,E1 -20778.267,E2 -20778.267} C_VEL
LIN {X 0,Y 283.068,Z 452.038,A -85,B 0,C 180,E1 -20780.649,E2 -20780.649} C_VEL
LIN {X 0,Y 287.089,Z 454.513,A -85,B 0,C 180,E1 -20782.262,E2 -20782.262} C_VEL
LIN {X 0,Y 289.941,Z 456.308,A -85,B 0,C 180,E1 -20783.617,E2 -20783.617} C_VEL
LIN {X 0,Y 293.345,Z 458.604,A -85,B 0,C 180,E1 -20785.878,E2 -20785.878} C_VEL
LIN {X 0,Y 295.473,Z 459.625,A -85,B 0,C 180,E1 -20787.409,E2 -20787.409} C_VEL
LIN {X 0,Y 296.767,Z 460.098,A -85,B 0,C 180,E1 -20788.643,E2 -20788.643} C_VEL
LIN {X 0,Y 297.66,Z 460.275,A -85,B 0,C 180,E1 -20790,E2 -20790} C_VEL
LIN {X 0,Y 296.736,Z 460.099,A -85,B 0,C 180,E1 -20791.357,E2 -20791.357} C_VEL
LIN {X 0,Y 295.229,Z 459.545,A -85,B 0,C 180,E1 -20792.729,E2 -20792.729} C_VEL
LIN {X 0,Y 293.293,Z 458.605,A -85,B 0,C 180,E1 -20794.122,E2 -20794.122} C_VEL
LIN {X 0,Y 289.941,Z 456.309,A -85,B 0,C 180,E1 -20796.383,E2 -20796.383} C_VEL
LIN {X 0,Y 287.057,Z 454.514,A -85,B 0,C 180,E1 -20797.739,E2 -20797.739} C_VEL
LIN {X 0,Y 281.161,Z 450.776,A -85,B 0,C 180,E1 -20800.077,E2 -20800.077} C_VEL
LIN {X 0,Y 273.727,Z 445.788,A -85,B 0,C 180,E1 -20802.672,E2 -20802.672} C_VEL
LIN {X 0,Y 265.5,Z 439.868,A -85,B 0,C 180,E1 -20805.35,E2 -20805.35} C_VEL
LIN {X 0,Y 255.795,Z 431.723,A -85,B 0,C 180,E1 -20808.581,E2 -20808.581} C_VEL
LIN {X 0,Y 248.614,Z 424.482,A -85,B 0,C 180,E1 -20811.117,E2 -20811.117} C_VEL
LIN {X 0,Y 241.858,Z 415.968,A -85,B 0,C 180,E1 -20813.751,E2 -20813.751} C_VEL
